LIN {X 0,Y 249.343,Z 705.614,A -85,B 0,C 180,E1 -25800.898,E2 -25800.898} C_VEL
LIN {X 0,Y 264.067,Z 715.978,A -85,B 0,C 180,E1 -25804.807,E2 -25804.807} C_VEL
LIN {X 0,Y 274.251,Z 722.94,A -85,B 0,C 180,E1 -25807.395,E2 -25807.395} C_VEL
LIN {X 0,Y 282.566,Z 728.902,A -85,B 0,C 180,E1 -25809.623,E2 -25809.623} C_VEL
LIN {X 0,Y 289.203,Z 733.495,A -85,B 0,C 180,E1 -25811.584,E2 -25811.584} C_VEL
LIN {X 0,Y 294.521,Z 737.29,A -85,B 0,C 180,E1 -25813.361,E2 -25813.361} C_VEL
LIN {X 0,Y 299.139,Z 740.278,A -85,B 0,C 180,E1 -25815.023,E2 -25815.023} C_VEL
LIN {X 0,Y 304.429,Z 743.64,A -85,B 0,C 180,E1 -25817.206,E2 -25817.206} C_VEL
LIN {X 0,Y 308.808,Z 746.666,A -85,B 0,C 180,E1 -25819.51,E2 -25819.51} C_VEL
LIN {X 0,Y 312.468,Z 748.873,A -85,B 0,C 180,E1 -25821.741,E2 -25821.741} C_VEL
LIN {X 0,Y 315.031,Z 750.212,A -85,B 0,C 180,E1 -25823.596,E2 -25823.596} C_VEL
LIN {X 0,Y 317.169,Z 751.257,A -85,B 0,C 180,E1 -25825.649,E2 -25825.649} C_VEL
LIN {X 0,Y 318.513,Z 751.721,A -85,B 0,C 180,E1 -25827.471,E2 -25827.471} C_VEL
LIN {X 0,Y 319.007,Z 751.919,A -85,B 0,C 180,E1 -25828.738,E2 -25828.738} C_VEL
LIN {X 0,Y 319.27,Z 751.929,A -85,B 0,C 180,E1 -25830,E2 -25830} C_VEL
LIN {X 0,Y 319.005,Z 751.919,A -85,B 0,C 180,E1 -25831.262,E2 -25831.262} C_VEL
LIN {X 0,Y 318.514,Z 751.721,A -85,B 0,C 180,E1 -25832.529,E2 -25832.529} C_VEL
LIN {X 0,Y 317.183,Z 751.226,A -85,B 0,C 180,E1 -25834.384,E2 -25834.384} C_VEL
LIN {X 0,Y 315.022,Z 750.196,A -85,B 0,C 180,E1 -25836.404,E2 -25836.404} C_VEL
LIN {X 0,Y 312.468,Z 748.905,A -85,B 0,C 180,E1 -25838.259,E2 -25838.259} C_VEL
LIN {X 0,Y 308.808,Z 746.698,A -85,B 0,C 180,E1 -25840.49,E2 -25840.49} C_VEL
LIN {X 0,Y 304.441,Z 743.645,A -85,B 0,C 180,E1 -25842.796,E2 -25842.796} C_VEL
LIN {X 0,Y 299.167,Z 740.269,A -85,B 0,C 180,E1 -25844.975,E2 -25844.975} C_VEL
LIN {X 0,Y 293.787,Z 736.797,A -85,B 0,C 180,E1 -25846.889,E2 -25846.889} C_VEL
LIN {X 0,Y 287.515,Z 732.243,A -85,B 0,C 180,E1 -25848.958,E2 -25848.958} C_VEL
LIN {X 0,Y 282.543,Z 728.898,A -85,B 0,C 180,E1 -25850.379,E2 -25850.379} C_VEL
LIN {X 0,Y 274.122,Z 722.857,A -85,B 0,C 180,E1 -25852.638,E2 -25852.638} C_VEL
LIN {X 0,Y 261.416,Z 714.087,A -85,B 0,C 180,E1 -25855.897,E2 -25855.897} C_VEL
LIN {X 0,Y 247.011,Z 703.927,A -85,B 0,C 180,E1 -25859.749,E2 -25859.749} C_VEL
LIN {X 0,Y 233.268,Z 692.779,A -85,B 0,C 180,E1 -25863.908,E2 -25863.908} C_VEL
LIN {X 0,Y 222.302,Z 681.729,A -85,B 0,C 180,E1 -25867.782,E2 -25867.782} C_VEL
LIN {X 0,Y 212.171,Z 669.521,A -85,B 0,C 180,E1 -25871.816,E2 -25871.816} C_VEL
LIN {X 0,Y 203.151,Z 656.416,A -85,B 0,C 180,E1 -25875.8,E2 -25875.8} C_VEL
LIN {X 0,Y 196.212,Z 644.549,A -85,B 0,C 180,E1 -25879.096,E2 -25879.096} C_VEL
LIN {X 0,Y 189.227,Z 630.541,A -85,B 0,C 180,E1 -25882.568,E2 -25882.568} C_VEL
LIN {X 0,Y 181.522,Z 611.257,A -85,B 0,C 180,E1 -25887.261,E2 -25887.261} C_VEL
LIN {X 0,Y 177.428,Z 602.179,A -85,B 0,C 180,E1 -25890.115,E2 -25890.115} C_VEL
LIN {X 0,Y 173.282,Z 594.104,A -85,B 0,C 180,E1 -25893.343,E2 -25893.343} C_VEL
LIN {X 0,Y 169.438,Z 587.347,A -85,B 0,C 180,E1 -25896.795,E2 -25896.795} C_VEL
LIN {X 0,Y 167.126,Z 583.517,A -85,B 0,C 180,E1 -25899.192,E2 -25899.192} C_VEL
LIN {X 0,Y 165.368,Z 580.676,A -85,B 0,C 180,E1 -25901.254,E2 -25901.254} C_VEL
LIN {X 0,Y 163.166,Z 577.17,A -85,B 0,C 180,E1 -25904.272,E2 -25904.272} C_VEL
LIN {X 0,Y 160.907,Z 573.312,A -85,B 0,C 180,E1 -25908.311,E2 -25908.311} C_VEL
LIN {X 0,Y 158.622,Z 569.898,A -85,B 0,C 180,E1 -25915.156,E2 -25915.156} C_VEL
LIN {X 0,Y 158.338,Z 568.536,A -85,B 0,C 180,E1 -25918.094,E2 -25918.094} C_VEL
LIN {X 0,Y 158.304,Z 568.373,A -85,B 0,C 180,E1 -25920.637,E2 -25920.637} C_VEL
LIN {X 0,Y 158.563,Z 569.545,A -85,B 0,C 180,E1 -25923.972,E2 -25923.972} C_VEL
LIN {X 0,Y 160.772,Z 573.178,A -85,B 0,C 180,E1 -25931.027,E2 -25931.027} C_VEL
LIN {X 0,Y 163.913,Z 578.324,A -85,B 0,C 180,E1 -25936.423,E2 -25936.423} C_VEL
LIN {X 0,Y 166.721,Z 582.763,A -85,B 0,C 180,E1 -25939.95,E2 -25939.95} C_VEL
LIN {X 0,Y 169.433,Z 587.305,A -85,B 0,C 180,E1 -25942.805,E2 -25942.805} C_VEL
LIN {X 0,Y 172.211,Z 592.35,A -85,B 0,C 180,E1 -25945.374,E2 -25945.374} C_VEL
LIN {X 0,Y 175.708,Z 601.255,A -85,B 0,C 180,E1 -25948.417,E2 -25948.417} C_VEL
LIN {X 0,Y 178.834,Z 610.413,A -85,B 0,C 180,E1 -25950.906,E2 -25950.906} C_VEL
LIN {X 0,Y 178.834,Z 612.491,A -85,B 0,C 180,E1 -25951.064,E2 -25951.064} C_VEL
LIN {X 0,Y 175.369,Z 650.601,A -85,B 0,C 180,E1 -25952.268,E2 -25952.268} C_VEL
LIN {X 0,Y 172.985,Z 664.836,A -85,B 0,C 180,E1 -25952.945,E2 -25952.945} C_VEL
LIN {X 0,Y 169.387,Z 678.905,A -85,B 0,C 180,E1 -25953.922,E2 -25953.922} C_VEL
LIN {X 0,Y 165.395,Z 691.016,A -85,B 0,C 180,E1 -25955.119,E2 -25955.119} C_VEL
LIN {X 0,Y 161.495,Z 700.931,A -85,B 0,C 180,E1 -25956.383,E2 -25956.383} C_VEL
LIN {X 0,Y 157.061,Z 710.649,A -85,B 0,C 180,E1 -25957.941,E2 -25957.941} C_VEL
LIN {X 0,Y 152.151,Z 720.062,A -85,B 0,C 180,E1 -25959.834,E2 -25959.834} C_VEL
LIN {X 0,Y 146.951,Z 729.125,A -85,B 0,C 180,E1 -25962.184,E2 -25962.184} C_VEL
LIN {X 0,Y 142.539,Z 736.054,A -85,B 0,C 180,E1 -25964.364,E2 -25964.364} C_VEL
LIN {X 0,Y 137.263,Z 743.572,A -85,B 0,C 180,E1 -25967.282,E2 -25967.282} C_VEL
LIN {X 0,Y 132.349,Z 750.042,A -85,B 0,C 180,E1 -25970.416,E2 -25970.416} C_VEL
LIN {X 0,Y 127.119,Z 756.583,A -85,B 0,C 180,E1 -25974.514,E2 -25974.514} C_VEL
LIN {X 0,Y 122.603,Z 762.018,A -85,B 0,C 180,E1 -25978.943,E2 -25978.943} C_VEL
LIN {X 0,Y 118.918,Z 766.47,A -85,B 0,C 180,E1 -25983.689,E2 -25983.689} C_VEL
LIN {X 0,Y 115.972,Z 770.022,A -85,B 0,C 180,E1 -25988.679,E2 -25988.679} C_VEL
LIN {X 0,Y 114.424,Z 771.967,A -85,B 0,C 180,E1 -25992.116,E2 -25992.116} C_VEL
LIN {X 0,Y 112.645,Z 774.671,A -85,B 0,C 180,E1 -25999.212,E2 -25999.212} C_VEL
LIN {X 0,Y 112.129,Z 775.98,A -85,B 0,C 180,E1 -26006.407,E2 -26006.407} C_VEL
LIN {X 0,Y 112.252,Z 776.239,A -85,B 0,C 180,E1 -26010,E2 -26010} C_VEL
LIN {X 0,Y 112.24,Z 775.497,A -85,B 0,C 180,E1 -26017.194,E2 -26017.194} C_VEL
LIN {X 0,Y 112.645,Z 774.671,A -85,B 0,C 180,E1 -26020.788,E2 -26020.788} C_VEL
LIN {X 0,Y 114.423,Z 771.967,A -85,B 0,C 180,E1 -26027.885,E2 -26027.885} C_VEL
LIN {X 0,Y 116.863,Z 769.003,A -85,B 0,C 180,E1 -26033.01,E2 -26033.01} C_VEL
LIN {X 0,Y 120.039,Z 765.169,A -85,B 0,C 180,E1 -26037.929,E2 -26037.929} C_VEL
LIN {X 0,Y 124.031,Z 760.401,A -85,B 0,C 180,E1 -26042.567,E2 -26042.567} C_VEL
LIN {X 0,Y 129.676,Z 753.456,A -85,B 0,C 180,E1 -26047.568,E2 -26047.568} C_VEL
LIN {X 0,Y 134.24,Z 747.582,A -85,B 0,C 180,E1 -26050.875,E2 -26050.875} C_VEL
LIN {X 0,Y 139.338,Z 740.737,A -85,B 0,C 180,E1 -26053.909,E2 -26053.909} C_VEL
LIN {X 0,Y 145.565,Z 731.458,A -85,B 0,C 180,E1 -26057.103,E2 -26057.103} C_VEL
LIN {X 0,Y 151.017,Z 722.182,A -85,B 0,C 180,E1 -26059.644,E2 -26059.644} C_VEL
LIN {X 0,Y 155.84,Z 713.129,A -85,B 0,C 180,E1 -26061.587,E2 -26061.587} C_VEL
LIN {X 0,Y 160.214,Z 703.858,A -85,B 0,C 180,E1 -26063.182,E2 -26063.182} C_VEL
LIN {X 0,Y 164.071,Z 694.521,A -85,B 0,C 180,E1 -26064.473,E2 -26064.473} C_VEL
LIN {X 0,Y 167.744,Z 684.271,A -85,B 0,C 180,E1 -26065.571,E2 -26065.571} C_VEL
LIN {X 0,Y 170.756,Z 673.982,A -85,B 0,C 180,E1 -26066.453,E2 -26066.453} C_VEL
LIN {X 0,Y 173.478,Z 662.099,A -85,B 0,C 180,E1 -26067.205,E2 -26067.205} C_VEL
LIN {X 0,Y 175.386,Z 650.33,A -85,B 0,C 180,E1 -26067.733,E2 -26067.733} C_VEL
LIN {X 0,Y 176.331,Z 641.978,A -85,B 0,C 180,E1 -26068.02,E2 -26068.02} C_VEL
LIN {X 0,Y 176.312,Z 638.104,A -85,B 0,C 180,E1 -26068.322,E2 -26068.322} C_VEL
LIN {X 0,Y 174.402,Z 626.17,A -85,B 0,C 180,E1 -26070.298,E2 -26070.298} C_VEL
LIN {X 0,Y 174.415,Z 622.295,A -85,B 0,C 180,E1 -26070.606,E2 -26070.606} C_VEL
LIN {X 0,Y 175.1,Z 613.268,A -85,B 0,C 180,E1 -26070.947,E2 -26070.947} C_VEL
LIN {X 0,Y 172.214,Z 604.583,A -85,B 0,C 180,E1 -26073.489,E2 -26073.489} C_VEL
LIN {X 0,Y 169.385,Z 597.046,A -85,B 0,C 180,E1 -26076.218,E2 -26076.218} C_VEL
LIN {X 0,Y 165.751,Z 590.516,A -85,B 0,C 180,E1 -26080.009,E2 -26080.009} C_VEL
LIN {X 0,Y 163.947,Z 587.5,A -85,B 0,C 180,E1 -26082.215,E2 -26082.215} C_VEL
LIN {X 0,Y 161.676,Z 583.716,A -85,B 0,C 180,E1 -26085.524,E2 -26085.524} C_VEL
LIN {X 0,Y 159.683,Z 580.121,A -85,B 0,C 180,E1 -26089.378,E2 -26089.378} C_VEL
LIN {X 0,Y 157.461,Z 575.531,A -85,B 0,C 180,E1 -26098.72,E2 -26098.72} C_VEL
LIN {X 0,Y 157.431,Z 575.384,A -85,B 0,C 180,E1 -26100.638,E2 -26100.638} C_VEL
LIN {X 0,Y 157.577,Z 576.308,A -85,B 0,C 180,E1 -26103.515,E2 -26103.515} C_VEL
LIN {X 0,Y 159.657,Z 580.101,A -85,B 0,C 180,E1 -26110.961,E2 -26110.961} C_VEL
LIN {X 0,Y 162.611,Z 585.221,A -85,B 0,C 180,E1 -26116.314,E2 -26116.314} C_VEL
LIN {X 0,Y 164.955,Z 589.145,A -85,B 0,C 180,E1 -26119.441,E2 -26119.441} C_VEL
LIN {X 0,Y 168.312,Z 595.05,A -85,B 0,C 180,E1 -26123.127,E2 -26123.127} C_VEL
LIN {X 0,Y 172.251,Z 602.608,A -85,B 0,C 180,E1 -26126.748,E2 -26126.748} C_VEL
LIN {X 0,Y 176.372,Z 611.496,A -85,B 0,C 180,E1 -26130.034,E2 -26130.034} C_VEL
LIN {X 0,Y 180.211,Z 621.162,A -85,B 0,C 180,E1 -26132.804,E2 -26132.804} C_VEL
LIN {X 0,Y 186.639,Z 637.619,A -85,B 0,C 180,E1 -26136.823,E2 -26136.823} C_VEL
LIN {X 0,Y 193.199,Z 651.318,A -85,B 0,C 180,E1 -26140.47,E2 -26140.47} C_VEL
LIN {X 0,Y 199.834,Z 663.107,A -85,B 0,C 180,E1 -26143.993,E2 -26143.993} C_VEL
LIN {X 0,Y 206.871,Z 673.757,A -85,B 0,C 180,E1 -26147.454,E2 -26147.454} C_VEL
LIN {X 0,Y 215.839,Z 684.961,A -85,B 0,C 180,E1 -26151.394,E2 -26151.394} C_VEL
LIN {X 0,Y 224.654,Z 694.377,A -85,B 0,C 180,E1 -26154.852,E2 -26154.852} C_VEL
LIN {X 0,Y 234.457,Z 702.998,A -85,B 0,C 180,E1 -26158.209,E2 -26158.209} C_VEL
LIN {X 0,Y 248.506,Z 713.424,A -85,B 0,C 180,E1 -26162.414,E2 -26162.414} C_VEL
LIN {X 0,Y 259.962,Z 721.098,A -85,B 0,C 180,E1 -26165.528,E2 -26165.528} C_VEL
LIN {X 0,Y 270.032,Z 727.797,A -85,B 0,C 180,E1 -26168.198,E2 -26168.198} C_VEL
LIN {X 0,Y 280.047,Z 734.699,A -85,B 0,C 180,E1 -26170.959,E2 -26170.959} C_VEL
LIN {X 0,Y 286.565,Z 739.311,A -85,B 0,C 180,E1 -26173.03,E2 -26173.03} C_VEL
LIN {X 0,Y 292.618,Z 743.324,A -85,B 0,C 180,E1 -26175.152,E2 -26175.152} C_VEL
LIN {X 0,Y 296.251,Z 745.63,A -85,B 0,C 180,E1 -26176.565,E2 -26176.565} C_VEL
LIN {X 0,Y 298.933,Z 747.459,A -85,B 0,C 180,E1 -26177.785,E2 -26177.785} C_VEL
LIN {X 0,Y 301.745,Z 749.392,A -85,B 0,C 180,E1 -26179.262,E2 -26179.262} C_VEL
LIN {X 0,Y 305.564,Z 751.769,A -85,B 0,C 180,E1 -26181.49,E2 -26181.49} C_VEL
LIN {X 0,Y 308.374,Z 753.28,A -85,B 0,C 180,E1 -26183.457,E2 -26183.457} C_VEL
LIN {X 0,Y 310.322,Z 754.209,A -85,B 0,C 180,E1 -26185.187,E2 -26185.187} C_VEL
LIN {X 0,Y 311.213,Z 754.584,A -85,B 0,C 180,E1 -26186.115,E2 -26186.115} C_VEL
LIN {X 0,Y 312.139,Z 754.94,A -85,B 0,C 180,E1 -26187.419,E2 -26187.419} C_VEL
LIN {X 0,Y 312.683,Z 755.143,A -85,B 0,C 180,E1 -26188.712,E2 -26188.712} C_VEL
LIN {X 0,Y 312.947,Z 755.169,A -85,B 0,C 180,E1 -26190,E2 -26190} C_VEL
LIN {X 0,Y 312.681,Z 755.141,A -85,B 0,C 180,E1 -26191.288,E2 -26191.288} C_VEL
LIN {X 0,Y 312.138,Z 754.937,A -85,B 0,C 180,E1 -26192.581,E2 -26192.581} C_VEL
LIN {X 0,Y 310.329,Z 754.212,A -85,B 0,C 180,E1 -26194.83,E2 -26194.83} C_VEL
LIN {X 0,Y 308.364,Z 753.256,A -85,B 0,C 180,E1 -26196.543,E2 -26196.543} C_VEL
LIN {X 0,Y 305.57,Z 751.76,A -85,B 0,C 180,E1 -26198.519,E2 -26198.519} C_VEL
LIN {X 0,Y 300.901,Z 748.83,A -85,B 0,C 180,E1 -26201.199,E2 -26201.199} C_VEL
LIN {X 0,Y 298.945,Z 747.432,A -85,B 0,C 180,E1 -26202.215,E2 -26202.215} C_VEL
LIN {X 0,Y 295.517,Z 745.126,A -85,B 0,C 180,E1 -26203.758,E2 -26203.758} C_VEL
LIN {X 0,Y 289.867,Z 741.603,A -85,B 0,C 180,E1 -26205.837,E2 -26205.837} C_VEL
LIN {X 0,Y 283.245,Z 736.916,A -85,B 0,C 180,E1 -26208.091,E2 -26208.091} C_VEL
LIN {X 0,Y 276.681,Z 732.425,A -85,B 0,C 180,E1 -26209.978,E2 -26209.978} C_VEL
LIN {X 0,Y 268.367,Z 726.639,A -85,B 0,C 180,E1 -26212.263,E2 -26212.263} C_VEL
LIN {X 0,Y 256.678,Z 718.841,A -85,B 0,C 180,E1 -26215.372,E2 -26215.372} C_VEL
LIN {X 0,Y 241.269,Z 708.265,A -85,B 0,C 180,E1 -26219.682,E2 -26219.682} C_VEL
LIN {X 0,Y 227.281,Z 696.899,A -85,B 0,C 180,E1 -26224.193,E2 -26224.193} C_VEL
LIN {X 0,Y 217.681,Z 687.148,A -85,B 0,C 180,E1 -26227.837,E2 -26227.837} C_VEL
LIN {X 0,Y 209.331,Z 676.985,A -85,B 0,C 180,E1 -26231.427,E2 -26231.427} C_VEL
LIN {X 0,Y 202.538,Z 667.322,A -85,B 0,C 180,E1 -26234.657,E2 -26234.657} C_VEL
LIN {X 0,Y 195.897,Z 656.31,A -85,B 0,C 180,E1 -26238.069,E2 -26238.069} C_VEL
LIN {X 0,Y 190.345,Z 645.491,A -85,B 0,C 180,E1 -26241.122,E2 -26241.122} C_VEL
LIN {X 0,Y 184.465,Z 632.548,A -85,B 0,C 180,E1 -26244.428,E2 -26244.428} C_VEL
LIN {X 0,Y 178.246,Z 615.988,A -85,B 0,C 180,E1 -26248.589,E2 -26248.589} C_VEL
LIN {X 0,Y 174.561,Z 607.48,A -85,B 0,C 180,E1 -26251.358,E2 -26251.358} C_VEL
LIN {X 0,Y 170.911,Z 599.958,A -85,B 0,C 180,E1 -26254.419,E2 -26254.419} C_VEL
LIN {X 0,Y 167.054,Z 592.841,A -85,B 0,C 180,E1 -26258.167,E2 -26258.167} C_VEL
LIN {X 0,Y 164.13,Z 587.743,A -85,B 0,C 180,E1 -26261.593,E2 -26261.593} C_VEL
LIN {X 0,Y 161.728,Z 583.787,A -85,B 0,C 180,E1 -26265.049,E2 -26265.049} C_VEL
LIN {X 0,Y 159.558,Z 580.057,A -85,B 0,C 180,E1 -26269.239,E2 -26269.239} C_VEL
LIN {X 0,Y 157.469,Z 575.62,A -85,B 0,C 180,E1 -26278.083,E2 -26278.083} C_VEL
LIN {X 0,Y 157.438,Z 575.431,A -85,B 0,C 180,E1 -26280.641,E2 -26280.641} C_VEL
LIN {X 0,Y 157.623,Z 576.478,A -85,B 0,C 180,E1 -26283.516,E2 -26283.516} C_VEL
LIN {X 0,Y 159.886,Z 580.526,A -85,B 0,C 180,E1 -26291.089,E2 -26291.089} C_VEL
LIN {X 0,Y 162.452,Z 584.977,A -85,B 0,C 180,E1 -26295.688,E2 -26295.688} C_VEL
LIN {X 0,Y 165.069,Z 589.338,A -85,B 0,C 180,E1 -26299.187,E2 -26299.187} C_VEL
LIN {X 0,Y 168.093,Z 594.615,A -85,B 0,C 180,E1 -26302.51,E2 -26302.51} C_VEL
LIN {X 0,Y 169.951,Z 598.44,A -85,B 0,C 180,E1 -26304.347,E2 -26304.347} C_VEL
LIN {X 0,Y 173.054,Z 607.008,A -85,B 0,C 180,E1 -26307.273,E2 -26307.273} C_VEL
LIN {X 0,Y 175.104,Z 613.293,A -85,B 0,C 180,E1 -26309.058,E2 -26309.058} C_VEL
LIN {X 0,Y 172.897,Z 639.291,A -85,B 0,C 180,E1 -26309.905,E2 -26309.905} C_VEL
LIN {X 0,Y 170.844,Z 656.23,A -85,B 0,C 180,E1 -26310.507,E2 -26310.507} C_VEL
LIN {X 0,Y 168.29,Z 668.57,A -85,B 0,C 180,E1 -26311.168,E2 -26311.168} C_VEL
LIN {X 0,Y 165.182,Z 679.779,A -85,B 0,C 180,E1 -26311.977,E2 -26311.977} C_VEL
LIN {X 0,Y 161.404,Z 690.818,A -85,B 0,C 180,E1 -26313.052,E2 -26313.052} C_VEL
LIN {X 0,Y 157.387,Z 700.733,A -85,B 0,C 180,E1 -26314.302,E2 -26314.302} C_VEL
LIN {X 0,Y 152.795,Z 710.451,A -85,B 0,C 180,E1 -26315.839,E2 -26315.839} C_VEL
LIN {X 0,Y 147.696,Z 719.863,A -85,B 0,C 180,E1 -26317.714,E2 -26317.714} C_VEL
LIN {X 0,Y 142.813,Z 728.023,A -85,B 0,C 180,E1 -26319.775,E2 -26319.775} C_VEL
LIN {X 0,Y 137.633,Z 735.854,A -85,B 0,C 180,E1 -26322.234,E2 -26322.234} C_VEL
LIN {X 0,Y 132.114,Z 743.374,A -85,B 0,C 180,E1 -26325.183,E2 -26325.183} C_VEL
LIN {X 0,Y 126.909,Z 749.843,A -85,B 0,C 180,E1 -26328.354,E2 -26328.354} C_VEL
LIN {X 0,Y 121.375,Z 756.383,A -85,B 0,C 180,E1 -26332.557,E2 -26332.557} C_VEL
LIN {X 0,Y 116.524,Z 761.818,A -85,B 0,C 180,E1 -26337.125,E2 -26337.125} C_VEL
LIN {X 0,Y 112.55,Z 766.27,A -85,B 0,C 180,E1 -26342.075,E2 -26342.075} C_VEL
LIN {X 0,Y 109.341,Z 769.822,A -85,B 0,C 180,E1 -26347.316,E2 -26347.316} C_VEL
LIN {X 0,Y 107.64,Z 771.767,A -85,B 0,C 180,E1 -26350.946,E2 -26350.946} C_VEL
LIN {X 0,Y 105.636,Z 774.471,A -85,B 0,C 180,E1 -26358.487,E2 -26358.487} C_VEL
LIN {X 0,Y 105.036,Z 775.781,A -85,B 0,C 180,E1 -26366.164,E2 -26366.164} C_VEL
LIN {X 0,Y 105.17,Z 776.042,A -85,B 0,C 180,E1 -26370,E2 -26370} C_VEL
LIN {X 0,Y 105.175,Z 775.299,A -85,B 0,C 180,E1 -26377.68,E2 -26377.68} C_VEL
LIN {X 0,Y 105.636,Z 774.471,A -85,B 0,C 180,E1 -26381.513,E2 -26381.513} C_VEL
LIN {X 0,Y 107.639,Z 771.767,A -85,B 0,C 180,E1 -26389.054,E2 -26389.054} C_VEL
LIN {X 0,Y 110.319,Z 768.804,A -85,B 0,C 180,E1 -26394.461,E2 -26394.461} C_VEL
LIN {X 0,Y 114.989,Z 763.502,A -85,B 0,C 180,E1 -26401.164,E2 -26401.164} C_VEL
LIN {X 0,Y 119.675,Z 758.297,A -85,B 0,C 180,E1 -26405.962,E2 -26405.962} C_VEL
LIN {X 0,Y 125.011,Z 752.119,A -85,B 0,C 180,E1 -26410.279,E2 -26410.279} C_VEL
LIN {X 0,Y 129.955,Z 746.046,A -85,B 0,C 180,E1 -26413.591,E2 -26413.591} C_VEL
LIN {X 0,Y 135.408,Z 738.978,A -85,B 0,C 180,E1 -26416.604,E2 -26416.604} C_VEL
LIN {X 0,Y 139.995,Z 732.521,A -85,B 0,C 180,E1 -26418.852,E2 -26418.852} C_VEL
LIN {X 0,Y 145.902,Z 723.043,A -85,B 0,C 180,E1 -26421.512,E2 -26421.512} C_VEL
LIN {X 0,Y 150.886,Z 714.17,A -85,B 0,C 180,E1 -26423.461,E2 -26423.461} C_VEL
LIN {X 0,Y 155.409,Z 705.124,A -85,B 0,C 180,E1 -26425.049,E2 -26425.049} C_VEL
LIN {X 0,Y 160.05,Z 694.323,A -85,B 0,C 180,E1 -26426.543,E2 -26426.543} C_VEL
LIN {X 0,Y 163.841,Z 684.073,A -85,B 0,C 180,E1 -26427.616,E2 -26427.616} C_VEL
LIN {X 0,Y 167.251,Z 672.563,A -85,B 0,C 180,E1 -26428.568,E2 -26428.568} C_VEL
LIN {X 0,Y 169.814,Z 661.454,A -85,B 0,C 180,E1 -26429.247,E2 -26429.247} C_VEL
LIN {X 0,Y 171.692,Z 650.197,A -85,B 0,C 180,E1 -26429.735,E2 -26429.735} C_VEL
LIN {X 0,Y 174.415,Z 622.295,A -85,B 0,C 180,E1 -26430.606,E2 -26430.606} C_VEL
LIN {X 0,Y 174.31,Z 619.282,A -85,B 0,C 180,E1 -26430.914,E2 -26430.914} C_VEL
LIN {X 0,Y 173.654,Z 616.695,A -85,B 0,C 180,E1 -26431.52,E2 -26431.52} C_VEL
LIN {X 0,Y 172.484,Z 614.168,A -85,B 0,C 180,E1 -26432.459,E2 -26432.459} C_VEL
LIN {X 0,Y 169.273,Z 608.739,A -85,B 0,C 180,E1 -26435.131,E2 -26435.131} C_VEL
LIN {X 0,Y 168.904,Z 607.826,A -85,B 0,C 180,E1 -26435.49,E2 -26435.49} C_VEL
LIN {X 0,Y 166.942,Z 602.523,A -85,B 0,C 180,E1 -26437.571,E2 -26437.571} C_VEL
LIN {X 0,Y 163.858,Z 596.656,A -85,B 0,C 180,E1 -26441.072,E2 -26441.072} C_VEL
LIN {X 0,Y 162.062,Z 593.514,A -85,B 0,C 180,E1 -26443.464,E2 -26443.464} C_VEL
LIN {X 0,Y 160.334,Z 590.422,A -85,B 0,C 180,E1 -26446.21,E2 -26446.21} C_VEL
LIN {X 0,Y 158.463,Z 586.917,A -85,B 0,C 180,E1 -26450.103,E2 -26450.103} C_VEL
LIN {X 0,Y 156.591,Z 582.617,A -85,B 0,C 180,E1 -26458.713,E2 -26458.713} C_VEL
LIN {X 0,Y 156.566,Z 582.432,A -85,B 0,C 180,E1 -26460.642,E2 -26460.642} C_VEL
LIN {X 0,Y 156.67,Z 583.317,A -85,B 0,C 180,E1 -26463.213,E2 -26463.213} C_VEL
LIN {X 0,Y 158.726,Z 587.386,A -85,B 0,C 180,E1 -26470.923,E2 -26470.923} C_VEL
LIN {X 0,Y 161.217,Z 591.969,A -85,B 0,C 180,E1 -26475.647,E2 -26475.647} C_VEL
LIN {X 0,Y 163.355,Z 595.768,A -85,B 0,C 180,E1 -26478.685,E2 -26478.685} C_VEL
LIN {X 0,Y 166.273,Z 601.159,A -85,B 0,C 180,E1 -26482.107,E2 -26482.107} C_VEL
LIN {X 0,Y 170.28,Z 609.336,A -85,B 0,C 180,E1 -26486.033,E2 -26486.033} C_VEL
LIN {X 0,Y 173.891,Z 617.792,A -85,B 0,C 180,E1 -26489.107,E2 -26489.107} C_VEL
LIN {X 0,Y 177.053,Z 626.293,A -85,B 0,C 180,E1 -26491.564,E2 -26491.564} C_VEL
LIN {X 0,Y 182.955,Z 642.316,A -85,B 0,C 180,E1 -26495.636,E2 -26495.636} C_VEL
LIN {X 0,Y 187.829,Z 653.466,A -85,B 0,C 180,E1 -26498.739,E2 -26498.739} C_VEL
LIN {X 0,Y 192.706,Z 663.195,A -85,B 0,C 180,E1 -26501.725,E2 -26501.725} C_VEL
LIN {X 0,Y 198.541,Z 673.231,A -85,B 0,C 180,E1 -26505.068,E2 -26505.068} C_VEL
LIN {X 0,Y 205.646,Z 683.514,A -85,B 0,C 180,E1 -26508.75,E2 -26508.75} C_VEL
LIN {X 0,Y 215.102,Z 694.784,A -85,B 0,C 180,E1 -26513.058,E2 -26513.058} C_VEL
LIN {X 0,Y 225.755,Z 704.956,A -85,B 0,C 180,E1 -26517.195,E2 -26517.195} C_VEL
LIN {X 0,Y 239.524,Z 715.344,A -85,B 0,C 180,E1 -26521.67,E2 -26521.67} C_VEL
LIN {X 0,Y 252.118,Z 723.619,A -85,B 0,C 180,E1 -26525.284,E2 -26525.284} C_VEL
LIN {X 0,Y 264.183,Z 731.336,A -85,B 0,C 180,E1 -26528.604,E2 -26528.604} C_VEL
LIN {X 0,Y 274.26,Z 738.006,A -85,B 0,C 180,E1 -26531.463,E2 -26531.463} C_VEL
LIN {X 0,Y 281.399,Z 743.034,A -85,B 0,C 180,E1 -26533.734,E2 -26533.734} C_VEL
LIN {X 0,Y 287.297,Z 746.886,A -85,B 0,C 180,E1 -26535.841,E2 -26535.841} C_VEL
LIN {X 0,Y 291.26,Z 749.46,A -85,B 0,C 180,E1 -26537.458,E2 -26537.458} C_VEL
LIN {X 0,Y 294.436,Z 751.63,A -85,B 0,C 180,E1 -26538.992,E2 -26538.992} C_VEL
LIN {X 0,Y 298.569,Z 754.255,A -85,B 0,C 180,E1 -26541.348,E2 -26541.348} C_VEL
LIN {X 0,Y 301.468,Z 755.905,A -85,B 0,C 180,E1 -26543.306,E2 -26543.306} C_VEL
LIN {X 0,Y 303.4,Z 756.816,A -85,B 0,C 180,E1 -26544.9,E2 -26544.9} C_VEL
LIN {X 0,Y 304.532,Z 757.314,A -85,B 0,C 180,E1 -26546.03,E2 -26546.03} C_VEL
LIN {X 0,Y 305.54,Z 757.724,A -85,B 0,C 180,E1 -26547.363,E2 -26547.363} C_VEL
LIN {X 0,Y 306.138,Z 757.962,A -85,B 0,C 180,E1 -26548.685,E2 -26548.685} C_VEL
LIN {X 0,Y 306.436,Z 757.996,A -85,B 0,C 180,E1 -26550,E2 -26550} C_VEL
LIN {X 0,Y 306.136,Z 757.958,A -85,B 0,C 180,E1 -26551.315,E2 -26551.315} C_VEL
LIN {X 0,Y 305.54,Z 757.717,A -85,B 0,C 180,E1 -26552.637,E2 -26552.637} C_VEL
LIN {X 0,Y 304.539,Z 757.299,A -85,B 0,C 180,E1 -26553.97,E2 -26553.97} C_VEL
LIN {X 0,Y 303.157,Z 756.7,A -85,B 0,C 180,E1 -26555.321,E2 -26555.321} C_VEL
LIN {X 0,Y 301.457,Z 755.888,A -85,B 0,C 180,E1 -26556.694,E2 -26556.694} C_VEL
LIN {X 0,Y 298.573,Z 754.251,A -85,B 0,C 180,E1 -26558.657,E2 -26558.657} C_VEL
LIN {X 0,Y 293.848,Z 751.22,A -85,B 0,C 180,E1 -26561.309,E2 -26561.309} C_VEL
LIN {X 0,Y 289.102,Z 747.988,A -85,B 0,C 180,E1 -26563.499,E2 -26563.499} C_VEL
LIN {X 0,Y 282.522,Z 743.805,A -85,B 0,C 180,E1 -26565.88,E2 -26565.88} C_VEL
LIN {X 0,Y 277.007,Z 739.833,A -85,B 0,C 180,E1 -26567.725,E2 -26567.725} C_VEL
LIN {X 0,Y 269.191,Z 734.697,A -85,B 0,C 180,E1 -26569.971,E2 -26569.971} C_VEL
LIN {X 0,Y 261.624,Z 729.69,A -85,B 0,C 180,E1 -26572.091,E2 -26572.091} C_VEL
LIN {X 0,Y 249.205,Z 721.757,A -85,B 0,C 180,E1 -26575.52,E2 -26575.52} C_VEL
LIN {X 0,Y 234.812,Z 712.009,A -85,B 0,C 180,E1 -26579.777,E2 -26579.777} C_VEL
LIN {X 0,Y 223.585,Z 703.071,A -85,B 0,C 180,E1 -26583.596,E2 -26583.596} C_VEL
LIN {X 0,Y 212.297,Z 691.665,A -85,B 0,C 180,E1 -26588.167,E2 -26588.167} C_VEL
LIN {X 0,Y 202.026,Z 678.57,A -85,B 0,C 180,E1 -26593.07,E2 -26593.07} C_VEL
LIN {X 0,Y 195.156,Z 667.699,A -85,B 0,C 180,E1 -26596.826,E2 -26596.826} C_VEL
LIN {X 0,Y 188.992,Z 655.999,A -85,B 0,C 180,E1 -26600.524,E2 -26600.524} C_VEL
LIN {X 0,Y 183.42,Z 643.374,A -85,B 0,C 180,E1 -26604.103,E2 -26604.103} C_VEL
LIN {X 0,Y 175.122,Z 620.901,A -85,B 0,C 180,E1 -26609.92,E2 -26609.92} C_VEL
LIN {X 0,Y 171.908,Z 613.017,A -85,B 0,C 180,E1 -26612.537,E2 -26612.537} C_VEL
LIN {X 0,Y 168.575,Z 605.761,A -85,B 0,C 180,E1 -26615.551,E2 -26615.551} C_VEL
LIN {X 0,Y 164.934,Z 598.64,A -85,B 0,C 180,E1 -26619.385,E2 -26619.385} C_VEL
LIN {X 0,Y 162.232,Z 593.761,A -85,B 0,C 180,E1 -26622.836,E2 -26622.836} C_VEL
LIN {X 0,Y 160.43,Z 590.565,A -85,B 0,C 180,E1 -26625.655,E2 -26625.655} C_VEL
LIN {X 0,Y 158.427,Z 586.931,A -85,B 0,C 180,E1 -26629.78,E2 -26629.78} C_VEL
LIN {X 0,Y 156.599,Z 582.705,A -85,B 0,C 180,E1 -26638.072,E2 -26638.072} C_VEL
LIN {X 0,Y 156.571,Z 582.488,A -85,B 0,C 180,E1 -26640.644,E2 -26640.644} C_VEL
LIN {X 0,Y 156.738,Z 583.696,A -85,B 0,C 180,E1 -26643.536,E2 -26643.536} C_VEL
LIN {X 0,Y 158.726,Z 587.364,A -85,B 0,C 180,E1 -26650.525,E2 -26650.525} C_VEL
LIN {X 0,Y 161.064,Z 591.729,A -85,B 0,C 180,E1 -26655.017,E2 -26655.017} C_VEL
LIN {X 0,Y 163.36,Z 595.761,A -85,B 0,C 180,E1 -26658.297,E2 -26658.297} C_VEL
LIN {X 0,Y 166.071,Z 600.746,A -85,B 0,C 180,E1 -26661.493,E2 -26661.493} C_VEL
LIN {X 0,Y 167.75,Z 604.501,A -85,B 0,C 180,E1 -26663.291,E2 -26663.291} C_VEL
LIN {X 0,Y 170.89,Z 613.943,A -85,B 0,C 180,E1 -26666.486,E2 -26666.486} C_VEL
LIN {X 0,Y 171.548,Z 616.124,A -85,B 0,C 180,E1 -26667.115,E2 -26667.115} C_VEL
LIN {X 0,Y 168.204,Z 650.359,A -85,B 0,C 180,E1 -26668.183,E2 -26668.183} C_VEL
LIN {X 0,Y 165.58,Z 665.008,A -85,B 0,C 180,E1 -26668.849,E2 -26668.849} C_VEL
LIN {X 0,Y 161.54,Z 679.582,A -85,B 0,C 180,E1 -26669.844,E2 -26669.844} C_VEL
LIN {X 0,Y 157.648,Z 690.62,A -85,B 0,C 180,E1 -26670.89,E2 -26670.89} C_VEL
LIN {X 0,Y 153.499,Z 700.535,A -85,B 0,C 180,E1 -26672.112,E2 -26672.112} C_VEL
LIN {X 0,Y 148.739,Z 710.252,A -85,B 0,C 180,E1 -26673.615,E2 -26673.615} C_VEL
LIN {X 0,Y 143.44,Z 719.664,A -85,B 0,C 180,E1 -26675.458,E2 -26675.458} C_VEL
LIN {X 0,Y 137.88,Z 728.532,A -85,B 0,C 180,E1 -26677.711,E2 -26677.711} C_VEL
LIN {X 0,Y 132.941,Z 735.655,A -85,B 0,C 180,E1 -26679.956,E2 -26679.956} C_VEL
LIN {X 0,Y 127.137,Z 743.174,A -85,B 0,C 180,E1 -26682.91,E2 -26682.91} C_VEL
LIN {X 0,Y 121.657,Z 749.643,A -85,B 0,C 180,E1 -26686.115,E2 -26686.115} C_VEL
LIN {X 0,Y 115.781,Z 756.184,A -85,B 0,C 180,E1 -26690.406,E2 -26690.406} C_VEL
LIN {X 0,Y 110.59,Z 761.619,A -85,B 0,C 180,E1 -26695.114,E2 -26695.114} C_VEL
LIN {X 0,Y 106.285,Z 766.071,A -85,B 0,C 180,E1 -26700.27,E2 -26700.27} C_VEL
LIN {X 0,Y 102.786,Z 769.623,A -85,B 0,C 180,E1 -26705.78,E2 -26705.78} C_VEL
LIN {X 0,Y 100.907,Z 771.568,A -85,B 0,C 180,E1 -26709.621,E2 -26709.621} C_VEL
LIN {X 0,Y 98.659,Z 774.273,A -85,B 0,C 180,E1 -26717.661,E2 -26717.661} C_VEL
LIN {X 0,Y 97.939,Z 775.583,A -85,B 0,C 180,E1 -26725.885,E2 -26725.885} C_VEL
LIN {X 0,Y 98.076,Z 775.844,A -85,B 0,C 180,E1 -26730,E2 -26730} C_VEL
LIN {X 0,Y 98.113,Z 775.1,A -85,B 0,C 180,E1 -26738.237,E2 -26738.237} C_VEL
LIN {X 0,Y 98.659,Z 774.273,A -85,B 0,C 180,E1 -26742.339,E2 -26742.339} C_VEL
LIN {X 0,Y 100.905,Z 771.568,A -85,B 0,C 180,E1 -26750.38,E2 -26750.38} C_VEL
LIN {X 0,Y 103.842,Z 768.604,A -85,B 0,C 180,E1 -26756.098,E2 -26756.098} C_VEL
LIN {X 0,Y 108.508,Z 763.74,A -85,B 0,C 180,E1 -26762.645,E2 -26762.645} C_VEL
LIN {X 0,Y 113.956,Z 758.097,A -85,B 0,C 180,E1 -26768.077,E2 -26768.077} C_VEL
LIN {X 0,Y 119.655,Z 751.92,A -85,B 0,C 180,E1 -26772.489,E2 -26772.489} C_VEL
LIN {X 0,Y 124.891,Z 745.847,A -85,B 0,C 180,E1 -26775.846,E2 -26775.846} C_VEL
LIN {X 0,Y 130.61,Z 738.779,A -85,B 0,C 180,E1 -26778.878,E2 -26778.878} C_VEL
LIN {X 0,Y 136.399,Z 730.885,A -85,B 0,C 180,E1 -26781.541,E2 -26781.541} C_VEL
LIN {X 0,Y 142.19,Z 721.784,A -85,B 0,C 180,E1 -26784.032,E2 -26784.032} C_VEL
LIN {X 0,Y 147.418,Z 712.732,A -85,B 0,C 180,E1 -26785.926,E2 -26785.926} C_VEL
LIN {X 0,Y 152.11,Z 703.461,A -85,B 0,C 180,E1 -26787.478,E2 -26787.478} C_VEL
LIN {X 0,Y 156.244,Z 694.125,A -85,B 0,C 180,E1 -26788.717,E2 -26788.717} C_VEL
LIN {X 0,Y 160.143,Z 683.875,A -85,B 0,C 180,E1 -26789.767,E2 -26789.767} C_VEL
LIN {X 0,Y 163.568,Z 672.726,A -85,B 0,C 180,E1 -26790.663,E2 -26790.663} C_VEL
LIN {X 0,Y 166.227,Z 661.622,A -85,B 0,C 180,E1 -26791.33,E2 -26791.33} C_VEL
LIN {X 0,Y 168.23,Z 650.049,A -85,B 0,C 180,E1 -26791.815,E2 -26791.815} C_VEL
LIN {X 0,Y 171.543,Z 616.171,A -85,B 0,C 180,E1 -26792.884,E2 -26792.884} C_VEL
LIN {X 0,Y 168.904,Z 607.826,A -85,B 0,C 180,E1 -26795.49,E2 -26795.49} C_VEL
LIN {X 0,Y 167.839,Z 605.596,A -85,B 0,C 180,E1 -26796.525,E2 -26796.525} C_VEL
LIN {X 0,Y 165.977,Z 603.346,A -85,B 0,C 180,E1 -26798.291,E2 -26798.291} C_VEL
LIN {X 0,Y 162.796,Z 601.308,A -85,B 0,C 180,E1 -26801.542,E2 -26801.542} C_VEL
LIN {X 0,Y 160.137,Z 599.18,A -85,B 0,C 180,E1 -26804.955,E2 -26804.955} C_VEL
LIN {X 0,Y 159.723,Z 598.508,A -85,B 0,C 180,E1 -26805.628,E2 -26805.628} C_VEL
LIN {X 0,Y 158.523,Z 596.35,A -85,B 0,C 180,E1 -26807.842,E2 -26807.842} C_VEL
LIN {X 0,Y 157.335,Z 593.765,A -85,B 0,C 180,E1 -26810.68,E2 -26810.68} C_VEL
LIN {X 0,Y 155.707,Z 589.528,A -85,B 0,C 180,E1 -26819.352,E2 -26819.352} C_VEL
LIN {X 0,Y 155.717,Z 589.698,A -85,B 0,C 180,E1 -26821.615,E2 -26821.615} C_VEL
LIN {X 0,Y 157.588,Z 594.287,A -85,B 0,C 180,E1 -26830.379,E2 -26830.379} C_VEL
LIN {X 0,Y 159.717,Z 598.395,A -85,B 0,C 180,E1 -26834.736,E2 -26834.736} C_VEL
LIN {X 0,Y 161.861,Z 602.537,A -85,B 0,C 180,E1 -26838.02,E2 -26838.02} C_VEL
LIN {X 0,Y 164.608,Z 608.014,A -85,B 0,C 180,E1 -26841.442,E2 -26841.442} C_VEL
LIN {X 0,Y 167.774,Z 614.812,A -85,B 0,C 180,E1 -26844.764,E2 -26844.764} C_VEL
LIN {X 0,Y 171.007,Z 622.869,A -85,B 0,C 180,E1 -26847.761,E2 -26847.761} C_VEL
LIN {X 0,Y 173.831,Z 630.857,A -85,B 0,C 180,E1 -26850.148,E2 -26850.148} C_VEL
LIN {X 0,Y 178.567,Z 644.992,A -85,B 0,C 180,E1 -26853.854,E2 -26853.854} C_VEL
LIN {X 0,Y 182.278,Z 654.564,A -85,B 0,C 180,E1 -26856.62,E2 -26856.62} C_VEL
LIN {X 0,Y 185.925,Z 663.197,A -85,B 0,C 180,E1 -26859.282,E2 -26859.282} C_VEL
LIN {X 0,Y 191.704,Z 674.574,A -85,B 0,C 180,E1 -26863.186,E2 -26863.186} C_VEL
LIN {X 0,Y 197.684,Z 684.259,A -85,B 0,C 180,E1 -26866.785,E2 -26866.785} C_VEL
LIN {X 0,Y 204.913,Z 693.824,A -85,B 0,C 180,E1 -26870.596,E2 -26870.596} C_VEL
LIN {X 0,Y 213.49,Z 703.305,A -85,B 0,C 180,E1 -26874.562,E2 -26874.562} C_VEL
LIN {X 0,Y 223.025,Z 711.686,A -85,B 0,C 180,E1 -26878.3,E2 -26878.3} C_VEL
LIN {X 0,Y 236.874,Z 721.516,A -85,B 0,C 180,E1 -26882.883,E2 -26882.883} C_VEL
LIN {X 0,Y 247.884,Z 728.415,A -85,B 0,C 180,E1 -26886.121,E2 -26886.121} C_VEL
LIN {X 0,Y 259.347,Z 735.421,A -85,B 0,C 180,E1 -26889.373,E2 -26889.373} C_VEL
LIN {X 0,Y 269.288,Z 741.658,A -85,B 0,C 180,E1 -26892.282,E2 -26892.282} C_VEL
LIN {X 0,Y 274.563,Z 745.246,A -85,B 0,C 180,E1 -26893.973,E2 -26893.973} C_VEL
LIN {X 0,Y 281.827,Z 750.023,A -85,B 0,C 180,E1 -26896.542,E2 -26896.542} C_VEL
LIN {X 0,Y 286.722,Z 753.247,A -85,B 0,C 180,E1 -26898.692,E2 -26898.692} C_VEL
LIN {X 0,Y 289.602,Z 755.254,A -85,B 0,C 180,E1 -26900.22,E2 -26900.22} C_VEL
LIN {X 0,Y 292.187,Z 756.765,A -85,B 0,C 180,E1 -26901.702,E2 -26901.702} C_VEL
LIN {X 0,Y 294.345,Z 758.043,A -85,B 0,C 180,E1 -26903.144,E2 -26903.144} C_VEL
LIN {X 0,Y 296.408,Z 759.071,A -85,B 0,C 180,E1 -26904.764,E2 -26904.764} C_VEL
LIN {X 0,Y 297.666,Z 759.613,A -85,B 0,C 180,E1 -26905.938,E2 -26905.938} C_VEL
LIN {X 0,Y 298.756,Z 760.057,A -85,B 0,C 180,E1 -26907.303,E2 -26907.303} C_VEL
LIN {X 0,Y 299.406,Z 760.324,A -85,B 0,C 180,E1 -26908.655,E2 -26908.655} C_VEL
LIN {X 0,Y 299.739,Z 760.376,A -85,B 0,C 180,E1 -26910,E2 -26910} C_VEL
LIN {X 0,Y 299.404,Z 760.318,A -85,B 0,C 180,E1 -26911.345,E2 -26911.345} C_VEL
LIN {X 0,Y 298.757,Z 760.046,A -85,B 0,C 180,E1 -26912.697,E2 -26912.697} C_VEL
LIN {X 0,Y 297.672,Z 759.593,A -85,B 0,C 180,E1 -26914.062,E2 -26914.062} C_VEL
LIN {X 0,Y 296.165,Z 758.946,A -85,B 0,C 180,E1 -26915.447,E2 -26915.447} C_VEL
LIN {X 0,Y 294.34,Z 758.049,A -85,B 0,C 180,E1 -26916.856,E2 -26916.856} C_VEL
LIN {X 0,Y 291.505,Z 756.375,A -85,B 0,C 180,E1 -26918.71,E2 -26918.71} C_VEL
LIN {X 0,Y 288.284,Z 754.315,A -85,B 0,C 180,E1 -26920.535,E2 -26920.535} C_VEL
LIN {X 0,Y 283.237,Z 750.87,A -85,B 0,C 180,E1 -26922.904,E2 -26922.904} C_VEL
LIN {X 0,Y 278.658,Z 747.985,A -85,B 0,C 180,E1 -26924.608,E2 -26924.608} C_VEL
LIN {X 0,Y 271.824,Z 743.306,A -85,B 0,C 180,E1 -26926.939,E2 -26926.939} C_VEL
LIN {X 0,Y 263.561,Z 738.072,A -85,B 0,C 180,E1 -26929.398,E2 -26929.398} C_VEL
LIN {X 0,Y 254.111,Z 732.241,A -85,B 0,C 180,E1 -26932.104,E2 -26932.104} C_VEL
LIN {X 0,Y 244.171,Z 726.129,A -85,B 0,C 180,E1 -26934.953,E2 -26934.953} C_VEL
LIN {X 0,Y 227.514,Z 715.124,A -85,B 0,C 180,E1 -26940.127,E2 -26940.127} C_VEL
LIN {X 0,Y 216.628,Z 706.265,A -85,B 0,C 180,E1 -26944.141,E2 -26944.141} C_VEL
LIN {X 0,Y 207.6,Z 697.044,A -85,B 0,C 180,E1 -26948.086,E2 -26948.086} C_VEL
LIN {X 0,Y 199.396,Z 686.716,A -85,B 0,C 180,E1 -26952.255,E2 -26952.255} C_VEL
LIN {X 0,Y 193.65,Z 677.893,A -85,B 0,C 180,E1 -26955.606,E2 -26955.606} C_VEL
LIN {X 0,Y 188.155,Z 667.755,A -85,B 0,C 180,E1 -26959.183,E2 -26959.183} C_VEL
LIN {X 0,Y 183.329,Z 657.227,A -85,B 0,C 180,E1 -26962.6,E2 -26962.6} C_VEL
LIN {X 0,Y 178.743,Z 645.328,A -85,B 0,C 180,E1 -26966.065,E2 -26966.065} C_VEL
LIN {X 0,Y 172.056,Z 625.631,A -85,B 0,C 180,E1 -26971.34,E2 -26971.34} C_VEL
LIN {X 0,Y 168.774,Z 617.189,A -85,B 0,C 180,E1 -26974.273,E2 -26974.273} C_VEL
LIN {X 0,Y 165.401,Z 609.599,A -85,B 0,C 180,E1 -26977.682,E2 -26977.682} C_VEL
LIN {X 0,Y 162.362,Z 603.464,A -85,B 0,C 180,E1 -26981.312,E2 -26981.312} C_VEL
LIN {X 0,Y 160.41,Z 599.794,A -85,B 0,C 180,E1 -26984.109,E2 -26984.109} C_VEL
LIN {X 0,Y 158.946,Z 597.009,A -85,B 0,C 180,E1 -26986.643,E2 -26986.643} C_VEL
LIN {X 0,Y 157.365,Z 593.853,A -85,B 0,C 180,E1 -26990.198,E2 -26990.198} C_VEL
LIN {X 0,Y 155.708,Z 589.614,A -85,B 0,C 180,E1 -26998.708,E2 -26998.708} C_VEL
LIN {X 0,Y 155.704,Z 589.551,A -85,B 0,C 180,E1 -27000.648,E2 -27000.648} C_VEL
LIN {X 0,Y 155.897,Z 591.052,A -85,B 0,C 180,E1 -27003.879,E2 -27003.879} C_VEL
LIN {X 0,Y 157.576,Z 594.253,A -85,B 0,C 180,E1 -27009.953,E2 -27009.953} C_VEL
LIN {X 0,Y 159.656,Z 598.375,A -85,B 0,C 180,E1 -27014.256,E2 -27014.256} C_VEL
LIN {X 0,Y 161.693,Z 602.171,A -85,B 0,C 180,E1 -27017.388,E2 -27017.388} C_VEL
LIN {X 0,Y 164.216,Z 607.182,A -85,B 0,C 180,E1 -27020.595,E2 -27020.595} C_VEL
LIN {X 0,Y 165.54,Z 610.425,A -85,B 0,C 180,E1 -27022.136,E2 -27022.136} C_VEL
LIN {X 0,Y 168.128,Z 618.919,A -85,B 0,C 180,E1 -27025.04,E2 -27025.04} C_VEL
LIN {X 0,Y 164.959,Z 650.223,A -85,B 0,C 180,E1 -27026.009,E2 -27026.009} C_VEL
LIN {X 0,Y 162.22,Z 665.081,A -85,B 0,C 180,E1 -27026.671,E2 -27026.671} C_VEL
LIN {X 0,Y 158.132,Z 679.384,A -85,B 0,C 180,E1 -27027.616,E2 -27027.616} C_VEL
LIN {X 0,Y 154.116,Z 690.421,A -85,B 0,C 180,E1 -27028.62,E2 -27028.62} C_VEL
LIN {X 0,Y 149.839,Z 700.336,A -85,B 0,C 180,E1 -27029.808,E2 -27029.808} C_VEL
LIN {X 0,Y 144.927,Z 710.054,A -85,B 0,C 180,E1 -27031.276,E2 -27031.276} C_VEL
LIN {X 0,Y 139.435,Z 719.466,A -85,B 0,C 180,E1 -27033.077,E2 -27033.077} C_VEL
LIN {X 0,Y 134.025,Z 727.8,A -85,B 0,C 180,E1 -27035.145,E2 -27035.145} C_VEL
LIN {X 0,Y 128.482,Z 735.456,A -85,B 0,C 180,E1 -27037.52,E2 -27037.52} C_VEL
LIN {X 0,Y 122.392,Z 742.975,A -85,B 0,C 180,E1 -27040.463,E2 -27040.463} C_VEL
LIN {X 0,Y 116.614,Z 749.444,A -85,B 0,C 180,E1 -27043.682,E2 -27043.682} C_VEL
LIN {X 0,Y 110.356,Z 755.984,A -85,B 0,C 180,E1 -27048.035,E2 -27048.035} C_VEL
LIN {X 0,Y 104.811,Z 761.419,A -85,B 0,C 180,E1 -27052.881,E2 -27052.881} C_VEL
LIN {X 0,Y 100.118,Z 765.871,A -85,B 0,C 180,E1 -27058.233,E2 -27058.233} C_VEL
LIN {X 0,Y 96.317,Z 769.424,A -85,B 0,C 180,E1 -27064.037,E2 -27064.037} C_VEL
LIN {X 0,Y 94.241,Z 771.369,A -85,B 0,C 180,E1 -27068.108,E2 -27068.108} C_VEL
LIN {X 0,Y 91.687,Z 774.073,A -85,B 0,C 180,E1 -27076.706,E2 -27076.706} C_VEL
LIN {X 0,Y 90.837,Z 775.384,A -85,B 0,C 180,E1 -27085.563,E2 -27085.563} C_VEL
LIN {X 0,Y 90.975,Z 775.646,A -85,B 0,C 180,E1 -27090,E2 -27090} C_VEL
LIN {X 0,Y 91.078,Z 774.901,A -85,B 0,C 180,E1 -27098.878,E2 -27098.878} C_VEL
LIN {X 0,Y 91.687,Z 774.073,A -85,B 0,C 180,E1 -27103.294,E2 -27103.294} C_VEL
LIN {X 0,Y 94.24,Z 771.369,A -85,B 0,C 180,E1 -27111.893,E2 -27111.893} C_VEL
LIN {X 0,Y 98.73,Z 767.139,A -85,B 0,C 180,E1 -27119.886,E2 -27119.886} C_VEL
LIN {X 0,Y 102.957,Z 763.157,A -85,B 0,C 180,E1 -27125.226,E2 -27125.226} C_VEL
LIN {X 0,Y 108.423,Z 757.898,A -85,B 0,C 180,E1 -27130.405,E2 -27130.405} C_VEL
LIN {X 0,Y 114.483,Z 751.72,A -85,B 0,C 180,E1 -27134.907,E2 -27134.907} C_VEL
LIN {X 0,Y 120.038,Z 745.648,A -85,B 0,C 180,E1 -27138.286,E2 -27138.286} C_VEL
LIN {X 0,Y 126.028,Z 738.579,A -85,B 0,C 180,E1 -27141.324,E2 -27141.324} C_VEL
LIN {X 0,Y 131.822,Z 731.06,A -85,B 0,C 180,E1 -27143.852,E2 -27143.852} C_VEL
LIN {X 0,Y 138.119,Z 721.585,A -85,B 0,C 180,E1 -27146.429,E2 -27146.429} C_VEL
LIN {X 0,Y 143.551,Z 712.533,A -85,B 0,C 180,E1 -27148.28,E2 -27148.28} C_VEL
LIN {X 0,Y 148.402,Z 703.262,A -85,B 0,C 180,E1 -27149.799,E2 -27149.799} C_VEL
LIN {X 0,Y 152.677,Z 693.927,A -85,B 0,C 180,E1 -27150.996,E2 -27150.996} C_VEL
LIN {X 0,Y 156.681,Z 683.676,A -85,B 0,C 180,E1 -27152.015,E2 -27152.015} C_VEL
LIN {X 0,Y 160.114,Z 672.9,A -85,B 0,C 180,E1 -27152.849,E2 -27152.849} C_VEL
LIN {X 0,Y 163.008,Z 661.132,A -85,B 0,C 180,E1 -27153.529,E2 -27153.529} C_VEL
LIN {X 0,Y 165.004,Z 649.852,A -85,B 0,C 180,E1 -27153.982,E2 -27153.982} C_VEL
LIN {X 0,Y 168.131,Z 618.895,A -85,B 0,C 180,E1 -27154.96,E2 -27154.96} C_VEL
LIN {X 0,Y 165.355,Z 609.865,A -85,B 0,C 180,E1 -27158.084,E2 -27158.084} C_VEL
LIN {X 0,Y 163.785,Z 606.244,A -85,B 0,C 180,E1 -27159.922,E2 -27159.922} C_VEL
LIN {X 0,Y 161.065,Z 600.908,A -85,B 0,C 180,E1 -27163.522,E2 -27163.522} C_VEL
LIN {X 0,Y 159.723,Z 598.508,A -85,B 0,C 180,E1 -27165.628,E2 -27165.628} C_VEL
LIN {X 0,Y 158.936,Z 597.475,A -85,B 0,C 180,E1 -27166.961,E2 -27166.961} C_VEL
LIN {X 0,Y 158.131,Z 597.084,A -85,B 0,C 180,E1 -27168.349,E2 -27168.349} C_VEL
LIN {X 0,Y 156.644,Z 597.469,A -85,B 0,C 180,E1 -27171.196,E2 -27171.196} C_VEL
LIN {X 0,Y 155.498,Z 598.193,A -85,B 0,C 180,E1 -27174.124,E2 -27174.124} C_VEL
LIN {X 0,Y 154.996,Z 598.039,A -85,B 0,C 180,E1 -27176.338,E2 -27176.338} C_VEL
LIN {X 0,Y 154.914,Z 597.725,A -85,B 0,C 180,E1 -27177.069,E2 -27177.069} C_VEL
LIN {X 0,Y 154.841,Z 596.45,A -85,B 0,C 180,E1 -27179.999,E2 -27179.999} C_VEL
LIN {X 0,Y 154.852,Z 597.245,A -85,B 0,C 180,E1 -27182.356,E2 -27182.356} C_VEL
LIN {X 0,Y 156.474,Z 601.223,A -85,B 0,C 180,E1 -27189.859,E2 -27189.859} C_VEL
LIN {X 0,Y 158.362,Z 605.114,A -85,B 0,C 180,E1 -27194.018,E2 -27194.018} C_VEL
LIN {X 0,Y 160.463,Z 609.401,A -85,B 0,C 180,E1 -27197.441,E2 -27197.441} C_VEL
LIN {X 0,Y 163.242,Z 615.383,A -85,B 0,C 180,E1 -27201.082,E2 -27201.082} C_VEL
LIN {X 0,Y 166.254,Z 622.593,A -85,B 0,C 180,E1 -27204.408,E2 -27204.408} C_VEL
LIN {X 0,Y 169.05,Z 630.309,A -85,B 0,C 180,E1 -27207.153,E2 -27207.153} C_VEL
LIN {X 0,Y 171.997,Z 639.893,A -85,B 0,C 180,E1 -27209.849,E2 -27209.849} C_VEL
LIN {X 0,Y 176.07,Z 652.976,A -85,B 0,C 180,E1 -27213.541,E2 -27213.541} C_VEL
LIN {X 0,Y 180.21,Z 664.52,A -85,B 0,C 180,E1 -27217.19,E2 -27217.19} C_VEL
LIN {X 0,Y 184.892,Z 675.275,A -85,B 0,C 180,E1 -27220.971,E2 -27220.971} C_VEL
LIN {X 0,Y 190.037,Z 684.827,A -85,B 0,C 180,E1 -27224.639,E2 -27224.639} C_VEL
LIN {X 0,Y 196.542,Z 694.575,A -85,B 0,C 180,E1 -27228.669,E2 -27228.669} C_VEL
LIN {X 0,Y 205.631,Z 705.395,A -85,B 0,C 180,E1 -27233.446,E2 -27233.446} C_VEL
LIN {X 0,Y 215.798,Z 714.767,A -85,B 0,C 180,E1 -27237.858,E2 -27237.858} C_VEL
LIN {X 0,Y 229.411,Z 724.422,A -85,B 0,C 180,E1 -27242.672,E2 -27242.672} C_VEL
LIN {X 0,Y 241.56,Z 731.776,A -85,B 0,C 180,E1 -27246.41,E2 -27246.41} C_VEL
LIN {X 0,Y 254.14,Z 739.062,A -85,B 0,C 180,E1 -27250.089,E2 -27250.089} C_VEL
LIN {X 0,Y 263.632,Z 744.671,A -85,B 0,C 180,E1 -27252.948,E2 -27252.948} C_VEL
LIN {X 0,Y 269.485,Z 748.41,A -85,B 0,C 180,E1 -27254.883,E2 -27254.883} C_VEL
LIN {X 0,Y 274.573,Z 751.672,A -85,B 0,C 180,E1 -27256.682,E2 -27256.682} C_VEL
LIN {X 0,Y 278.703,Z 754.326,A -85,B 0,C 180,E1 -27258.362,E2 -27258.362} C_VEL
LIN {X 0,Y 281.932,Z 756.539,A -85,B 0,C 180,E1 -27259.951,E2 -27259.951} C_VEL
LIN {X 0,Y 284.65,Z 758.219,A -85,B 0,C 180,E1 -27261.481,E2 -27261.481} C_VEL
LIN {X 0,Y 286.987,Z 759.635,A -85,B 0,C 180,E1 -27262.967,E2 -27262.967} C_VEL
LIN {X 0,Y 289.371,Z 760.92,A -85,B 0,C 180,E1 -27264.721,E2 -27264.721} C_VEL
LIN {X 0,Y 290.62,Z 761.471,A -85,B 0,C 180,E1 -27265.84,E2 -27265.84} C_VEL
LIN {X 0,Y 291.801,Z 761.961,A -85,B 0,C 180,E1 -27267.239,E2 -27267.239} C_VEL
LIN {X 0,Y 292.538,Z 762.244,A -85,B 0,C 180,E1 -27268.623,E2 -27268.623} C_VEL
LIN {X 0,Y 292.902,Z 762.308,A -85,B 0,C 180,E1 -27270,E2 -27270} C_VEL
LIN {X 0,Y 292.537,Z 762.237,A -85,B 0,C 180,E1 -27271.377,E2 -27271.377} C_VEL
LIN {X 0,Y 291.802,Z 761.946,A -85,B 0,C 180,E1 -27272.761,E2 -27272.761} C_VEL
LIN {X 0,Y 290.624,Z 761.449,A -85,B 0,C 180,E1 -27274.16,E2 -27274.16} C_VEL
LIN {X 0,Y 288.984,Z 760.736,A -85,B 0,C 180,E1 -27275.582,E2 -27275.582} C_VEL
LIN {X 0,Y 286.997,Z 759.659,A -85,B 0,C 180,E1 -27277.033,E2 -27277.033} C_VEL
LIN {X 0,Y 284.366,Z 758.082,A -85,B 0,C 180,E1 -27278.672,E2 -27278.672} C_VEL
LIN {X 0,Y 281.958,Z 756.52,A -85,B 0,C 180,E1 -27280.048,E2 -27280.048} C_VEL
LIN {X 0,Y 278.731,Z 754.34,A -85,B 0,C 180,E1 -27281.637,E2 -27281.637} C_VEL
LIN {X 0,Y 274.488,Z 751.595,A -85,B 0,C 180,E1 -27283.36,E2 -27283.36} C_VEL
LIN {X 0,Y 266.879,Z 746.681,A -85,B 0,C 180,E1 -27286.018,E2 -27286.018} C_VEL
LIN {X 0,Y 262.508,Z 743.98,A -85,B 0,C 180,E1 -27287.405,E2 -27287.405} C_VEL
LIN {X 0,Y 251.598,Z 737.566,A -85,B 0,C 180,E1 -27290.65,E2 -27290.65} C_VEL
LIN {X 0,Y 239.212,Z 730.363,A -85,B 0,C 180,E1 -27294.287,E2 -27294.287} C_VEL
LIN {X 0,Y 224.723,Z 721.324,A -85,B 0,C 180,E1 -27298.877,E2 -27298.877} C_VEL
LIN {X 0,Y 213.68,Z 712.982,A -85,B 0,C 180,E1 -27302.999,E2 -27302.999} C_VEL
LIN {X 0,Y 202.785,Z 702.309,A -85,B 0,C 180,E1 -27307.961,E2 -27307.961} C_VEL
LIN {X 0,Y 193.227,Z 689.851,A -85,B 0,C 180,E1 -27313.33,E2 -27313.33} C_VEL
LIN {X 0,Y 186.311,Z 678.142,A -85,B 0,C 180,E1 -27317.968,E2 -27317.968} C_VEL
LIN {X 0,Y 181.507,Z 667.765,A -85,B 0,C 180,E1 -27321.72,E2 -27321.72} C_VEL
LIN {X 0,Y 177.112,Z 656.114,A -85,B 0,C 180,E1 -27325.508,E2 -27325.508} C_VEL
LIN {X 0,Y 173.489,Z 644.753,A -85,B 0,C 180,E1 -27328.828,E2 -27328.828} C_VEL
LIN {X 0,Y 169.182,Z 630.665,A -85,B 0,C 180,E1 -27332.727,E2 -27332.727} C_VEL
LIN {X 0,Y 166.489,Z 623.232,A -85,B 0,C 180,E1 -27335.348,E2 -27335.348} C_VEL
LIN {X 0,Y 163.844,Z 616.816,A -85,B 0,C 180,E1 -27338.205,E2 -27338.205} C_VEL
LIN {X 0,Y 161.268,Z 611.08,A -85,B 0,C 180,E1 -27341.427,E2 -27341.427} C_VEL
LIN {X 0,Y 159.034,Z 606.512,A -85,B 0,C 180,E1 -27344.789,E2 -27344.789} C_VEL
LIN {X 0,Y 157.691,Z 603.776,A -85,B 0,C 180,E1 -27347.283,E2 -27347.283} C_VEL
LIN {X 0,Y 156.189,Z 600.655,A -85,B 0,C 180,E1 -27350.94,E2 -27350.94} C_VEL
LIN {X 0,Y 154.839,Z 596.695,A -85,B 0,C 180,E1 -27358.701,E2 -27358.701} C_VEL
LIN {X 0,Y 154.843,Z 596.694,A -85,B 0,C 180,E1 -27360.976,E2 -27360.976} C_VEL
LIN {X 0,Y 156.443,Z 601.124,A -85,B 0,C 180,E1 -27369.373,E2 -27369.373} C_VEL
LIN {X 0,Y 158.277,Z 605.014,A -85,B 0,C 180,E1 -27373.482,E2 -27373.482} C_VEL
LIN {X 0,Y 160.298,Z 609.051,A -85,B 0,C 180,E1 -27376.805,E2 -27376.805} C_VEL
LIN {X 0,Y 162.871,Z 614.629,A -85,B 0,C 180,E1 -27380.252,E2 -27380.252} C_VEL
LIN {X 0,Y 164.955,Z 621.955,A -85,B 0,C 180,E1 -27382.922,E2 -27382.922} C_VEL
LIN {X 0,Y 161.953,Z 650.145,A -85,B 0,C 180,E1 -27383.753,E2 -27383.753} C_VEL
LIN {X 0,Y 159.071,Z 665.271,A -85,B 0,C 180,E1 -27384.408,E2 -27384.408} C_VEL
LIN {X 0,Y 154.972,Z 679.186,A -85,B 0,C 180,E1 -27385.291,E2 -27385.291} C_VEL
LIN {X 0,Y 150.84,Z 690.223,A -85,B 0,C 180,E1 -27386.249,E2 -27386.249} C_VEL
LIN {X 0,Y 146.432,Z 700.138,A -85,B 0,C 180,E1 -27387.392,E2 -27387.392} C_VEL
LIN {X 0,Y 141.368,Z 709.856,A -85,B 0,C 180,E1 -27388.813,E2 -27388.813} C_VEL
LIN {X 0,Y 135.67,Z 719.267,A -85,B 0,C 180,E1 -27390.549,E2 -27390.549} C_VEL
LIN {X 0,Y 129.77,Z 727.984,A -85,B 0,C 180,E1 -27392.684,E2 -27392.684} C_VEL
LIN {X 0,Y 124.276,Z 735.258,A -85,B 0,C 180,E1 -27394.917,E2 -27394.917} C_VEL
LIN {X 0,Y 117.895,Z 742.776,A -85,B 0,C 180,E1 -27397.829,E2 -27397.829} C_VEL
LIN {X 0,Y 111.802,Z 749.245,A -85,B 0,C 180,E1 -27401.034,E2 -27401.034} C_VEL
LIN {X 0,Y 105.143,Z 755.785,A -85,B 0,C 180,E1 -27405.426,E2 -27405.426} C_VEL
LIN {X 0,Y 99.203,Z 761.22,A -85,B 0,C 180,E1 -27410.388,E2 -27410.388} C_VEL
LIN {X 0,Y 94.102,Z 765.671,A -85,B 0,C 180,E1 -27415.936,E2 -27415.936} C_VEL
LIN {X 0,Y 89.948,Z 769.225,A -85,B 0,C 180,E1 -27422.044,E2 -27422.044} C_VEL
LIN {X 0,Y 87.658,Z 771.17,A -85,B 0,C 180,E1 -27426.368,E2 -27426.368} C_VEL
LIN {X 0,Y 84.756,Z 773.874,A -85,B 0,C 180,E1 -27435.596,E2 -27435.596} C_VEL
LIN {X 0,Y 83.759,Z 775.186,A -85,B 0,C 180,E1 -27445.187,E2 -27445.187} C_VEL
LIN {X 0,Y 83.881,Z 775.448,A -85,B 0,C 180,E1 -27450,E2 -27450} C_VEL
LIN {X 0,Y 84.039,Z 774.703,A -85,B 0,C 180,E1 -27459.628,E2 -27459.628} C_VEL
LIN {X 0,Y 84.756,Z 773.874,A -85,B 0,C 180,E1 -27464.404,E2 -27464.404} C_VEL
LIN {X 0,Y 87.656,Z 771.169,A -85,B 0,C 180,E1 -27473.633,E2 -27473.633} C_VEL
LIN {X 0,Y 92.6,Z 766.94,A -85,B 0,C 180,E1 -27482.091,E2 -27482.091} C_VEL
LIN {X 0,Y 97.202,Z 762.958,A -85,B 0,C 180,E1 -27487.658,E2 -27487.658} C_VEL
LIN {X 0,Y 103.071,Z 757.698,A -85,B 0,C 180,E1 -27492.988,E2 -27492.988} C_VEL
LIN {X 0,Y 109.521,Z 751.52,A -85,B 0,C 180,E1 -27497.556,E2 -27497.556} C_VEL
LIN {X 0,Y 115.42,Z 745.449,A -85,B 0,C 180,E1 -27500.926,E2 -27500.926} C_VEL
LIN {X 0,Y 121.69,Z 738.38,A -85,B 0,C 180,E1 -27503.952,E2 -27503.952} C_VEL
LIN {X 0,Y 127.98,Z 730.529,A -85,B 0,C 180,E1 -27506.537,E2 -27506.537} C_VEL
LIN {X 0,Y 133.616,Z 722.445,A -85,B 0,C 180,E1 -27508.727,E2 -27508.727} C_VEL
LIN {X 0,Y 139.24,Z 713.575,A -85,B 0,C 180,E1 -27510.535,E2 -27510.535} C_VEL
LIN {X 0,Y 144.232,Z 704.527,A -85,B 0,C 180,E1 -27512.025,E2 -27512.025} C_VEL
LIN {X 0,Y 149.367,Z 693.729,A -85,B 0,C 180,E1 -27513.376,E2 -27513.376} C_VEL
LIN {X 0,Y 153.486,Z 683.479,A -85,B 0,C 180,E1 -27514.349,E2 -27514.349} C_VEL
LIN {X 0,Y 156.901,Z 673.086,A -85,B 0,C 180,E1 -27515.127,E2 -27515.127} C_VEL
LIN {X 0,Y 159.929,Z 661.095,A -85,B 0,C 180,E1 -27515.804,E2 -27515.804} C_VEL
LIN {X 0,Y 162.023,Z 649.654,A -85,B 0,C 180,E1 -27516.233,E2 -27516.233} C_VEL
LIN {X 0,Y 164.932,Z 621.764,A -85,B 0,C 180,E1 -27517.117,E2 -27517.117} C_VEL
LIN {X 0,Y 162.77,Z 614.382,A -85,B 0,C 180,E1 -27519.874,E2 -27519.874} C_VEL
LIN {X 0,Y 160.35,Z 609.156,A -85,B 0,C 180,E1 -27523.119,E2 -27523.119} C_VEL
LIN {X 0,Y 158.712,Z 605.939,A -85,B 0,C 180,E1 -27525.723,E2 -27525.723} C_VEL
LIN {X 0,Y 157.487,Z 603.427,A -85,B 0,C 180,E1 -27528.088,E2 -27528.088} C_VEL
LIN {X 0,Y 156.223,Z 600.609,A -85,B 0,C 180,E1 -27531.266,E2 -27531.266} C_VEL
LIN {X 0,Y 154.914,Z 597.725,A -85,B 0,C 180,E1 -27537.069,E2 -27537.069} C_VEL
LIN {X 0,Y 154.778,Z 597.505,A -85,B 0,C 180,E1 -27538.503,E2 -27538.503} C_VEL
LIN {X 0,Y 154.564,Z 598.737,A -85,B 0,C 180,E1 -27540.635,E2 -27540.635} C_VEL
LIN {X 0,Y 154.417,Z 601.072,A -85,B 0,C 180,E1 -27542.675,E2 -27542.675} C_VEL
LIN {X 0,Y 154.458,Z 604.791,A -85,B 0,C 180,E1 -27545.424,E2 -27545.424} C_VEL
LIN {X 0,Y 154.822,Z 606.983,A -85,B 0,C 180,E1 -27547.554,E2 -27547.554} C_VEL
LIN {X 0,Y 155.034,Z 607.449,A -85,B 0,C 180,E1 -27548.289,E2 -27548.289} C_VEL
LIN {X 0,Y 155.57,Z 608.694,A -85,B 0,C 180,E1 -27549.916,E2 -27549.916} C_VEL
LIN {X 0,Y 157.018,Z 611.814,A -85,B 0,C 180,E1 -27553.26,E2 -27553.26} C_VEL
LIN {X 0,Y 158.889,Z 615.846,A -85,B 0,C 180,E1 -27556.553,E2 -27556.553} C_VEL
LIN {X 0,Y 161.499,Z 622.025,A -85,B 0,C 180,E1 -27560.257,E2 -27560.257} C_VEL
LIN {X 0,Y 164.006,Z 628.518,A -85,B 0,C 180,E1 -27563.255,E2 -27563.255} C_VEL
LIN {X 0,Y 166.651,Z 636.426,A -85,B 0,C 180,E1 -27566.08,E2 -27566.08} C_VEL
LIN {X 0,Y 170.861,Z 652.288,A -85,B 0,C 180,E1 -27570.656,E2 -27570.656} C_VEL
LIN {X 0,Y 173.934,Z 662.902,A -85,B 0,C 180,E1 -27574.009,E2 -27574.009} C_VEL
LIN {X 0,Y 177.474,Z 673.286,A -85,B 0,C 180,E1 -27577.629,E2 -27577.629} C_VEL
LIN {X 0,Y 182.072,Z 683.914,A -85,B 0,C 180,E1 -27581.746,E2 -27581.746} C_VEL
LIN {X 0,Y 188.048,Z 694.537,A -85,B 0,C 180,E1 -27586.261,E2 -27586.261} C_VEL
LIN {X 0,Y 195.188,Z 704.237,A -85,B 0,C 180,E1 -27590.725,E2 -27590.725} C_VEL
LIN {X 0,Y 202.535,Z 712.315,A -85,B 0,C 180,E1 -27594.63,E2 -27594.63} C_VEL
LIN {X 0,Y 212.858,Z 721.033,A -85,B 0,C 180,E1 -27599.141,E2 -27599.141} C_VEL
LIN {X 0,Y 224.947,Z 729.106,A -85,B 0,C 180,E1 -27603.507,E2 -27603.507} C_VEL
LIN {X 0,Y 237.085,Z 736.075,A -85,B 0,C 180,E1 -27607.334,E2 -27607.334} C_VEL
LIN {X 0,Y 246.556,Z 741.19,A -85,B 0,C 180,E1 -27610.159,E2 -27610.159} C_VEL
LIN {X 0,Y 256.82,Z 746.863,A -85,B 0,C 180,E1 -27613.29,E2 -27613.29} C_VEL
LIN {X 0,Y 263.695,Z 750.894,A -85,B 0,C 180,E1 -27615.593,E2 -27615.593} C_VEL
LIN {X 0,Y 270.244,Z 754.839,A -85,B 0,C 180,E1 -27617.992,E2 -27617.992} C_VEL
LIN {X 0,Y 273.912,Z 757.243,A -85,B 0,C 180,E1 -27619.654,E2 -27619.654} C_VEL
LIN {X 0,Y 277.188,Z 759.397,A -85,B 0,C 180,E1 -27621.422,E2 -27621.422} C_VEL
LIN {X 0,Y 279.435,Z 760.813,A -85,B 0,C 180,E1 -27622.776,E2 -27622.776} C_VEL
LIN {X 0,Y 282.287,Z 762.275,A -85,B 0,C 180,E1 -27624.778,E2 -27624.778} C_VEL
LIN {X 0,Y 283.381,Z 762.789,A -85,B 0,C 180,E1 -27625.733,E2 -27625.733} C_VEL
LIN {X 0,Y 284.7,Z 763.368,A -85,B 0,C 180,E1 -27627.17,E2 -27627.17} C_VEL
LIN {X 0,Y 285.548,Z 763.688,A -85,B 0,C 180,E1 -27628.59,E2 -27628.59} C_VEL
LIN {X 0,Y 285.957,Z 763.771,A -85,B 0,C 180,E1 -27630,E2 -27630} C_VEL
LIN {X 0,Y 285.547,Z 763.679,A -85,B 0,C 180,E1 -27631.41,E2 -27631.41} C_VEL
LIN {X 0,Y 284.702,Z 763.348,A -85,B 0,C 180,E1 -27632.83,E2 -27632.83} C_VEL
LIN {X 0,Y 283.401,Z 762.779,A -85,B 0,C 180,E1 -27634.266,E2 -27634.266} C_VEL
LIN {X 0,Y 281.601,Z 761.973,A -85,B 0,C 180,E1 -27635.729,E2 -27635.729} C_VEL
LIN {X 0,Y 279.437,Z 760.82,A -85,B 0,C 180,E1 -27637.224,E2 -27637.224} C_VEL
LIN {X 0,Y 276.898,Z 759.196,A -85,B 0,C 180,E1 -27638.759,E2 -27638.759} C_VEL
LIN {X 0,Y 272.222,Z 756.069,A -85,B 0,C 180,E1 -27641.176,E2 -27641.176} C_VEL
LIN {X 0,Y 270.3,Z 754.837,A -85,B 0,C 180,E1 -27642.005,E2 -27642.005} C_VEL
LIN {X 0,Y 263.7,Z 750.896,A -85,B 0,C 180,E1 -27644.407,E2 -27644.407} C_VEL
LIN {X 0,Y 256.832,Z 746.84,A -85,B 0,C 180,E1 -27646.719,E2 -27646.719} C_VEL
LIN {X 0,Y 245.792,Z 740.787,A -85,B 0,C 180,E1 -27650.067,E2 -27650.067} C_VEL
LIN {X 0,Y 234.955,Z 734.819,A -85,B 0,C 180,E1 -27653.342,E2 -27653.342} C_VEL
LIN {X 0,Y 217.947,Z 724.689,A -85,B 0,C 180,E1 -27658.926,E2 -27658.926} C_VEL
LIN {X 0,Y 206.571,Z 716.022,A -85,B 0,C 180,E1 -27663.496,E2 -27663.496} C_VEL
LIN {X 0,Y 196.931,Z 706.382,A -85,B 0,C 180,E1 -27668.269,E2 -27668.269} C_VEL
LIN {X 0,Y 190.153,Z 697.636,A -85,B 0,C 180,E1 -27672.339,E2 -27672.339} C_VEL
LIN {X 0,Y 184.412,Z 688.366,A -85,B 0,C 180,E1 -27676.392,E2 -27676.392} C_VEL
LIN {X 0,Y 179.565,Z 678.466,A -85,B 0,C 180,E1 -27680.405,E2 -27680.405} C_VEL
LIN {X 0,Y 175.92,Z 669.063,A -85,B 0,C 180,E1 -27683.897,E2 -27683.897} C_VEL
LIN {X 0,Y 172.161,Z 657.201,A -85,B 0,C 180,E1 -27687.855,E2 -27687.855} C_VEL
LIN {X 0,Y 168.866,Z 644.683,A -85,B 0,C 180,E1 -27691.565,E2 -27691.565} C_VEL
LIN {X 0,Y 166.22,Z 635.05,A -85,B 0,C 180,E1 -27694.362,E2 -27694.362} C_VEL
LIN {X 0,Y 163.631,Z 627.459,A -85,B 0,C 180,E1 -27697.174,E2 -27697.174} C_VEL
LIN {X 0,Y 160.939,Z 620.671,A -85,B 0,C 180,E1 -27700.473,E2 -27700.473} C_VEL
LIN {X 0,Y 158.587,Z 615.243,A -85,B 0,C 180,E1 -27703.921,E2 -27703.921} C_VEL
LIN {X 0,Y 156.565,Z 610.701,A -85,B 0,C 180,E1 -27707.71,E2 -27707.71} C_VEL
LIN {X 0,Y 155.096,Z 607.502,A -85,B 0,C 180,E1 -27711.533,E2 -27711.533} C_VEL
LIN {X 0,Y 153.961,Z 603.653,A -85,B 0,C 180,E1 -27719.347,E2 -27719.347} C_VEL
LIN {X 0,Y 153.966,Z 603.832,A -85,B 0,C 180,E1 -27720.982,E2 -27720.982} C_VEL
LIN {X 0,Y 155.328,Z 607.985,A -85,B 0,C 180,E1 -27728.785,E2 -27728.785} C_VEL
LIN {X 0,Y 157.006,Z 611.825,A -85,B 0,C 180,E1 -27732.852,E2 -27732.852} C_VEL
LIN {X 0,Y 158.702,Z 615.439,A -85,B 0,C 180,E1 -27735.863,E2 -27735.863} C_VEL
LIN {X 0,Y 160.816,Z 620.435,A -85,B 0,C 180,E1 -27738.978,E2 -27738.978} C_VEL
LIN {X 0,Y 161.985,Z 624.943,A -85,B 0,C 180,E1 -27740.689,E2 -27740.689} C_VEL
LIN {X 0,Y 159.226,Z 649.957,A -85,B 0,C 180,E1 -27741.415,E2 -27741.415} C_VEL
LIN {X 0,Y 156.293,Z 664.982,A -85,B 0,C 180,E1 -27742.033,E2 -27742.033} C_VEL
LIN {X 0,Y 152.076,Z 678.988,A -85,B 0,C 180,E1 -27742.874,E2 -27742.874} C_VEL
LIN {X 0,Y 147.842,Z 690.025,A -85,B 0,C 180,E1 -27743.784,E2 -27743.784} C_VEL
LIN {X 0,Y 143.305,Z 699.94,A -85,B 0,C 180,E1 -27744.87,E2 -27744.87} C_VEL
LIN {X 0,Y 138.08,Z 709.657,A -85,B 0,C 180,E1 -27746.226,E2 -27746.226} C_VEL
LIN {X 0,Y 132.187,Z 719.068,A -85,B 0,C 180,E1 -27747.886,E2 -27747.886} C_VEL
LIN {X 0,Y 126.321,Z 727.45,A -85,B 0,C 180,E1 -27749.865,E2 -27749.865} C_VEL
LIN {X 0,Y 120.345,Z 735.06,A -85,B 0,C 180,E1 -27752.139,E2 -27752.139} C_VEL
LIN {X 0,Y 113.67,Z 742.578,A -85,B 0,C 180,E1 -27754.995,E2 -27754.995} C_VEL
LIN {X 0,Y 107.247,Z 749.045,A -85,B 0,C 180,E1 -27758.154,E2 -27758.154} C_VEL
LIN {X 0,Y 100.183,Z 755.585,A -85,B 0,C 180,E1 -27762.559,E2 -27762.559} C_VEL
LIN {X 0,Y 93.791,Z 761.02,A -85,B 0,C 180,E1 -27767.594,E2 -27767.594} C_VEL
LIN {X 0,Y 88.195,Z 765.511,A -85,B 0,C 180,E1 -27773.388,E2 -27773.388} C_VEL
LIN {X 0,Y 83.676,Z 769.024,A -85,B 0,C 180,E1 -27779.739,E2 -27779.739} C_VEL
LIN {X 0,Y 81.173,Z 770.971,A -85,B 0,C 180,E1 -27784.349,E2 -27784.349} C_VEL
LIN {X 0,Y 77.87,Z 773.675,A -85,B 0,C 180,E1 -27794.291,E2 -27794.291} C_VEL
LIN {X 0,Y 76.663,Z 774.988,A -85,B 0,C 180,E1 -27804.74,E2 -27804.74} C_VEL
LIN {X 0,Y 76.778,Z 775.25,A -85,B 0,C 180,E1 -27810,E2 -27810} C_VEL
LIN {X 0,Y 77.009,Z 774.503,A -85,B 0,C 180,E1 -27820.517,E2 -27820.517} C_VEL
LIN {X 0,Y 77.87,Z 773.675,A -85,B 0,C 180,E1 -27825.709,E2 -27825.709} C_VEL
LIN {X 0,Y 81.171,Z 770.971,A -85,B 0,C 180,E1 -27835.652,E2 -27835.652} C_VEL
LIN {X 0,Y 86.626,Z 766.74,A -85,B 0,C 180,E1 -27844.604,E2 -27844.604} C_VEL
LIN {X 0,Y 91.835,Z 762.6,A -85,B 0,C 180,E1 -27850.577,E2 -27850.577} C_VEL
LIN {X 0,Y 97.963,Z 757.499,A -85,B 0,C 180,E1 -27855.84,E2 -27855.84} C_VEL
LIN {X 0,Y 104.825,Z 751.321,A -85,B 0,C 180,E1 -27860.444,E2 -27860.444} C_VEL
LIN {X 0,Y 111.06,Z 745.25,A -85,B 0,C 180,E1 -27863.786,E2 -27863.786} C_VEL
LIN {X 0,Y 117.631,Z 738.181,A -85,B 0,C 180,E1 -27866.765,E2 -27866.765} C_VEL
LIN {X 0,Y 123.618,Z 731.084,A -85,B 0,C 180,E1 -27869.069,E2 -27869.069} C_VEL
LIN {X 0,Y 130.071,Z 722.247,A -85,B 0,C 180,E1 -27871.402,E2 -27871.402} C_VEL
LIN {X 0,Y 135.882,Z 713.377,A -85,B 0,C 180,E1 -27873.148,E2 -27873.148} C_VEL
LIN {X 0,Y 141.038,Z 704.329,A -85,B 0,C 180,E1 -27874.576,E2 -27874.576} C_VEL
LIN {X 0,Y 146.316,Z 693.531,A -85,B 0,C 180,E1 -27875.868,E2 -27875.868} C_VEL
LIN {X 0,Y 150.537,Z 683.28,A -85,B 0,C 180,E1 -27876.797,E2 -27876.797} C_VEL
LIN {X 0,Y 154.23,Z 672.253,A -85,B 0,C 180,E1 -27877.561,E2 -27877.561} C_VEL
LIN {X 0,Y 157.125,Z 661.042,A -85,B 0,C 180,E1 -27878.156,E2 -27878.156} C_VEL
LIN {X 0,Y 159.251,Z 649.751,A -85,B 0,C 180,E1 -27878.563,E2 -27878.563} C_VEL
LIN {X 0,Y 162.007,Z 625.014,A -85,B 0,C 180,E1 -27879.281,E2 -27879.281} C_VEL
LIN {X 0,Y 160.642,Z 619.954,A -85,B 0,C 180,E1 -27881.267,E2 -27881.267} C_VEL
LIN {X 0,Y 158.44,Z 614.86,A -85,B 0,C 180,E1 -27884.564,E2 -27884.564} C_VEL
LIN {X 0,Y 156.304,Z 610.233,A -85,B 0,C 180,E1 -27888.662,E2 -27888.662} C_VEL
LIN {X 0,Y 155.125,Z 607.479,A -85,B 0,C 180,E1 -27891.86,E2 -27891.86} C_VEL
LIN {X 0,Y 153.973,Z 603.522,A -85,B 0,C 180,E1 -27899.999,E2 -27899.999} C_VEL
LIN {X 0,Y 153.97,Z 604.438,A -85,B 0,C 180,E1 -27902.37,E2 -27902.37} C_VEL
LIN {X 0,Y 155.034,Z 607.449,A -85,B 0,C 180,E1 -27908.289,E2 -27908.289} C_VEL
LIN {X 0,Y 155.687,Z 609.34,A -85,B 0,C 180,E1 -27910.332,E2 -27910.332} C_VEL
LIN {X 0,Y 156.29,Z 612.415,A -85,B 0,C 180,E1 -27912.187,E2 -27912.187} C_VEL
LIN {X 0,Y 158.651,Z 625.609,A -85,B 0,C 180,E1 -27917.754,E2 -27917.754} C_VEL
LIN {X 0,Y 161.117,Z 632.303,A -85,B 0,C 180,E1 -27921.174,E2 -27921.174} C_VEL
LIN {X 0,Y 163.404,Z 639.473,A -85,B 0,C 180,E1 -27923.956,E2 -27923.956} C_VEL
LIN {X 0,Y 165.592,Z 648.869,A -85,B 0,C 180,E1 -27926.82,E2 -27926.82} C_VEL
LIN {X 0,Y 168.387,Z 661.5,A -85,B 0,C 180,E1 -27930.748,E2 -27930.748} C_VEL
LIN {X 0,Y 171.57,Z 673.556,A -85,B 0,C 180,E1 -27934.992,E2 -27934.992} C_VEL
LIN {X 0,Y 175.817,Z 685.516,A -85,B 0,C 180,E1 -27939.758,E2 -27939.758} C_VEL
LIN {X 0,Y 180.904,Z 695.937,A -85,B 0,C 180,E1 -27944.368,E2 -27944.368} C_VEL
LIN {X 0,Y 186.874,Z 705.102,A -85,B 0,C 180,E1 -27948.776,E2 -27948.776} C_VEL
LIN {X 0,Y 193.672,Z 713.334,A -85,B 0,C 180,E1 -27952.97,E2 -27952.97} C_VEL
LIN {X 0,Y 202.7,Z 721.739,A -85,B 0,C 180,E1 -27957.533,E2 -27957.533} C_VEL
LIN {X 0,Y 214.367,Z 729.962,A -85,B 0,C 180,E1 -27962.273,E2 -27962.273} C_VEL
LIN {X 0,Y 228.81,Z 738.13,A -85,B 0,C 180,E1 -27967.138,E2 -27967.138} C_VEL
LIN {X 0,Y 238.937,Z 743.34,A -85,B 0,C 180,E1 -27970.257,E2 -27970.257} C_VEL
LIN {X 0,Y 246.676,Z 747.274,A -85,B 0,C 180,E1 -27972.635,E2 -27972.635} C_VEL
LIN {X 0,Y 254.477,Z 751.346,A -85,B 0,C 180,E1 -27975.148,E2 -27975.148} C_VEL
LIN {X 0,Y 261.277,Z 755.095,A -85,B 0,C 180,E1 -27977.574,E2 -27977.574} C_VEL
LIN {X 0,Y 265.659,Z 757.553,A -85,B 0,C 180,E1 -27979.328,E2 -27979.328} C_VEL
LIN {X 0,Y 269.98,Z 760.317,A -85,B 0,C 180,E1 -27981.565,E2 -27981.565} C_VEL
LIN {X 0,Y 271.706,Z 761.39,A -85,B 0,C 180,E1 -27982.569,E2 -27982.569} C_VEL
LIN {X 0,Y 275.174,Z 763.245,A -85,B 0,C 180,E1 -27984.906,E2 -27984.906} C_VEL
LIN {X 0,Y 277.508,Z 764.388,A -85,B 0,C 180,E1 -27987.097,E2 -27987.097} C_VEL
LIN {X 0,Y 278.469,Z 764.782,A -85,B 0,C 180,E1 -27988.554,E2 -27988.554} C_VEL
LIN {X 0,Y 278.942,Z 764.883,A -85,B 0,C 180,E1 -27990,E2 -27990} C_VEL
LIN {X 0,Y 278.469,Z 764.769,A -85,B 0,C 180,E1 -27991.446,E2 -27991.446} C_VEL
LIN {X 0,Y 277.514,Z 764.369,A -85,B 0,C 180,E1 -27992.903,E2 -27992.903} C_VEL
LIN {X 0,Y 275.175,Z 763.231,A -85,B 0,C 180,E1 -27995.096,E2 -27995.096} C_VEL
LIN {X 0,Y 271.691,Z 761.391,A -85,B 0,C 180,E1 -27997.431,E2 -27997.431} C_VEL
LIN {X 0,Y 267.414,Z 758.625,A -85,B 0,C 180,E1 -27999.836,E2 -27999.836} C_VEL
LIN {X 0,Y 264.905,Z 757.091,A -85,B 0,C 180,E1 -28001.007,E2 -28001.007} C_VEL
LIN {X 0,Y 259.68,Z 754.181,A -85,B 0,C 180,E1 -28003.021,E2 -28003.021} C_VEL
LIN {X 0,Y 251.897,Z 749.945,A -85,B 0,C 180,E1 -28005.734,E2 -28005.734} C_VEL
LIN {X 0,Y 242.787,Z 745.286,A -85,B 0,C 180,E1 -28008.567,E2 -28008.567} C_VEL
LIN {X 0,Y 231.339,Z 739.407,A -85,B 0,C 180,E1 -28012.095,E2 -28012.095} C_VEL
LIN {X 0,Y 216.162,Z 731.07,A -85,B 0,C 180,E1 -28017.076,E2 -28017.076} C_VEL
LIN {X 0,Y 204.097,Z 722.863,A -85,B 0,C 180,E1 -28021.835,E2 -28021.835} C_VEL
LIN {X 0,Y 193.666,Z 713.347,A -85,B 0,C 180,E1 -28027.028,E2 -28027.028} C_VEL
LIN {X 0,Y 185.327,Z 702.914,A -85,B 0,C 180,E1 -28032.315,E2 -28032.315} C_VEL
LIN {X 0,Y 178.941,Z 692.19,A -85,B 0,C 180,E1 -28037.353,E2 -28037.353} C_VEL
LIN {X 0,Y 173.867,Z 680.422,A -85,B 0,C 180,E1 -28042.348,E2 -28042.348} C_VEL
LIN {X 0,Y 170.639,Z 670.23,A -85,B 0,C 180,E1 -28046.221,E2 -28046.221} C_VEL
LIN {X 0,Y 167.592,Z 658.274,A -85,B 0,C 180,E1 -28050.293,E2 -28050.293} C_VEL
LIN {X 0,Y 164.864,Z 645.473,A -85,B 0,C 180,E1 -28054.176,E2 -28054.176} C_VEL
LIN {X 0,Y 163.038,Z 638.259,A -85,B 0,C 180,E1 -28056.473,E2 -28056.473} C_VEL
LIN {X 0,Y 160.767,Z 631.284,A -85,B 0,C 180,E1 -28059.28,E2 -28059.28} C_VEL
LIN {X 0,Y 158.283,Z 624.691,A -85,B 0,C 180,E1 -28062.811,E2 -28062.811} C_VEL
LIN {X 0,Y 156.276,Z 619.772,A -85,B 0,C 180,E1 -28066.333,E2 -28066.333} C_VEL
LIN {X 0,Y 155.01,Z 616.874,A -85,B 0,C 180,E1 -28069.138,E2 -28069.138} C_VEL
LIN {X 0,Y 154.018,Z 614.371,A -85,B 0,C 180,E1 -28072.133,E2 -28072.133} C_VEL
LIN {X 0,Y 153.092,Z 610.729,A -85,B 0,C 180,E1 -28079.344,E2 -28079.344} C_VEL
LIN {X 0,Y 153.092,Z 610.886,A -85,B 0,C 180,E1 -28080.823,E2 -28080.823} C_VEL
LIN {X 0,Y 154.236,Z 614.829,A -85,B 0,C 180,E1 -28088.198,E2 -28088.198} C_VEL
LIN {X 0,Y 155.605,Z 618.274,A -85,B 0,C 180,E1 -28091.881,E2 -28091.881} C_VEL
LIN {X 0,Y 157.363,Z 622.348,A -85,B 0,C 180,E1 -28095.276,E2 -28095.276} C_VEL
LIN {X 0,Y 158.914,Z 626.488,A -85,B 0,C 180,E1 -28097.785,E2 -28097.785} C_VEL
LIN {X 0,Y 159.274,Z 628.101,A -85,B 0,C 180,E1 -28098.405,E2 -28098.405} C_VEL
LIN {X 0,Y 156.595,Z 650.983,A -85,B 0,C 180,E1 -28099.039,E2 -28099.039} C_VEL
LIN {X 0,Y 153.172,Z 666.86,A -85,B 0,C 180,E1 -28099.674,E2 -28099.674} C_VEL
LIN {X 0,Y 149.464,Z 678.791,A -85,B 0,C 180,E1 -28100.37,E2 -28100.37} C_VEL
LIN {X 0,Y 145.119,Z 689.827,A -85,B 0,C 180,E1 -28101.213,E2 -28101.213} C_VEL
LIN {X 0,Y 140.462,Z 699.742,A -85,B 0,C 180,E1 -28102.238,E2 -28102.238} C_VEL
LIN {X 0,Y 135.085,Z 709.459,A -85,B 0,C 180,E1 -28103.516,E2 -28103.516} C_VEL
LIN {X 0,Y 129.021,Z 718.87,A -85,B 0,C 180,E1 -28105.099,E2 -28105.099} C_VEL
LIN {X 0,Y 122.418,Z 727.891,A -85,B 0,C 180,E1 -28107.151,E2 -28107.151} C_VEL
LIN {X 0,Y 116.645,Z 734.938,A -85,B 0,C 180,E1 -28109.205,E2 -28109.205} C_VEL
LIN {X 0,Y 109.745,Z 742.38,A -85,B 0,C 180,E1 -28111.951,E2 -28111.951} C_VEL
LIN {X 0,Y 102.993,Z 748.846,A -85,B 0,C 180,E1 -28115.032,E2 -28115.032} C_VEL
LIN {X 0,Y 95.507,Z 755.387,A -85,B 0,C 180,E1 -28119.409,E2 -28119.409} C_VEL
LIN {X 0,Y 88.646,Z 760.821,A -85,B 0,C 180,E1 -28124.478,E2 -28124.478} C_VEL
LIN {X 0,Y 83.006,Z 764.994,A -85,B 0,C 180,E1 -28129.892,E2 -28129.892} C_VEL
LIN {X 0,Y 77.566,Z 768.824,A -85,B 0,C 180,E1 -28137.069,E2 -28137.069} C_VEL
LIN {X 0,Y 74.807,Z 770.772,A -85,B 0,C 180,E1 -28141.983,E2 -28141.983} C_VEL
LIN {X 0,Y 71.006,Z 773.475,A -85,B 0,C 180,E1 -28152.727,E2 -28152.727} C_VEL
LIN {X 0,Y 69.576,Z 774.789,A -85,B 0,C 180,E1 -28164.203,E2 -28164.203} C_VEL
LIN {X 0,Y 69.673,Z 775.052,A -85,B 0,C 180,E1 -28170,E2 -28170} C_VEL
LIN {X 0,Y 70.014,Z 774.305,A -85,B 0,C 180,E1 -28181.581,E2 -28181.581} C_VEL
LIN {X 0,Y 71.006,Z 773.475,A -85,B 0,C 180,E1 -28187.273,E2 -28187.273} C_VEL
LIN {X 0,Y 74.805,Z 770.772,A -85,B 0,C 180,E1 -28198.018,E2 -28198.018} C_VEL
LIN {X 0,Y 80.821,Z 766.54,A -85,B 0,C 180,E1 -28207.495,E2 -28207.495} C_VEL
LIN {X 0,Y 86.532,Z 762.401,A -85,B 0,C 180,E1 -28213.657,E2 -28213.657} C_VEL
LIN {X 0,Y 93.134,Z 757.3,A -85,B 0,C 180,E1 -28218.99,E2 -28218.99} C_VEL
LIN {X 0,Y 100.415,Z 751.121,A -85,B 0,C 180,E1 -28223.597,E2 -28223.597} C_VEL
LIN {X 0,Y 106.998,Z 745.051,A -85,B 0,C 180,E1 -28226.871,E2 -28226.871} C_VEL
LIN {X 0,Y 113.882,Z 737.982,A -85,B 0,C 180,E1 -28229.764,E2 -28229.764} C_VEL
LIN {X 0,Y 119.596,Z 731.527,A -85,B 0,C 180,E1 -28231.817,E2 -28231.817} C_VEL
LIN {X 0,Y 126.809,Z 722.048,A -85,B 0,C 180,E1 -28234.235,E2 -28234.235} C_VEL
LIN {X 0,Y 132.828,Z 713.179,A -85,B 0,C 180,E1 -28235.88,E2 -28235.88} C_VEL
LIN {X 0,Y 138.138,Z 704.131,A -85,B 0,C 180,E1 -28237.238,E2 -28237.238} C_VEL
LIN {X 0,Y 143.554,Z 693.332,A -85,B 0,C 180,E1 -28238.46,E2 -28238.46} C_VEL
LIN {X 0,Y 147.881,Z 683.082,A -85,B 0,C 180,E1 -28239.328,E2 -28239.328} C_VEL
LIN {X 0,Y 151.518,Z 672.545,A -85,B 0,C 180,E1 -28240.016,E2 -28240.016} C_VEL
LIN {X 0,Y 154.717,Z 660.398,A -85,B 0,C 180,E1 -28240.62,E2 -28240.62} C_VEL
LIN {X 0,Y 156.693,Z 650.259,A -85,B 0,C 180,E1 -28240.96,E2 -28240.96} C_VEL
LIN {X 0,Y 159.274,Z 628.047,A -85,B 0,C 180,E1 -28241.602,E2 -28241.602} C_VEL
LIN {X 0,Y 158.505,Z 625.214,A -85,B 0,C 180,E1 -28242.864,E2 -28242.864} C_VEL
LIN {X 0,Y 156.477,Z 620.213,A -85,B 0,C 180,E1 -28246.338,E2 -28246.338} C_VEL
LIN {X 0,Y 154.879,Z 616.562,A -85,B 0,C 180,E1 -28249.871,E2 -28249.871} C_VEL
LIN {X 0,Y 153.948,Z 614.183,A -85,B 0,C 180,E1 -28252.787,E2 -28252.787} C_VEL
LIN {X 0,Y 153.105,Z 610.587,A -85,B 0,C 180,E1 -28259.999,E2 -28259.999} C_VEL
LIN {X 0,Y 153.296,Z 612.778,A -85,B 0,C 180,E1 -28264.642,E2 -28264.642} C_VEL
LIN {X 0,Y 154.257,Z 614.94,A -85,B 0,C 180,E1 -28268.679,E2 -28268.679} C_VEL
LIN {X 0,Y 155.696,Z 618.461,A -85,B 0,C 180,E1 -28272.47,E2 -28272.47} C_VEL
LIN {X 0,Y 157.429,Z 622.521,A -85,B 0,C 180,E1 -28275.784,E2 -28275.784} C_VEL
LIN {X 0,Y 158.651,Z 625.609,A -85,B 0,C 180,E1 -28277.754,E2 -28277.754} C_VEL
LIN {X 0,Y 159.541,Z 629.685,A -85,B 0,C 180,E1 -28279.271,E2 -28279.271} C_VEL
LIN {X 0,Y 160.584,Z 637.784,A -85,B 0,C 180,E1 -28281.302,E2 -28281.302} C_VEL
LIN {X 0,Y 161.6,Z 647.891,A -85,B 0,C 180,E1 -28283.623,E2 -28283.623} C_VEL
LIN {X 0,Y 162.047,Z 650.959,A -85,B 0,C 180,E1 -28284.526,E2 -28284.526} C_VEL
LIN {X 0,Y 163.922,Z 662.294,A -85,B 0,C 180,E1 -28288.138,E2 -28288.138} C_VEL
LIN {X 0,Y 166.194,Z 673.815,A -85,B 0,C 180,E1 -28292.249,E2 -28292.249} C_VEL
LIN {X 0,Y 168.927,Z 684.092,A -85,B 0,C 180,E1 -28296.358,E2 -28296.358} C_VEL
LIN {X 0,Y 172.493,Z 693.848,A -85,B 0,C 180,E1 -28300.683,E2 -28300.683} C_VEL
LIN {X 0,Y 177.462,Z 703.638,A -85,B 0,C 180,E1 -28305.466,E2 -28305.466} C_VEL
LIN {X 0,Y 183.414,Z 712.264,A -85,B 0,C 180,E1 -28310.026,E2 -28310.026} C_VEL
LIN {X 0,Y 192.168,Z 721.689,A -85,B 0,C 180,E1 -28315.371,E2 -28315.371} C_VEL
LIN {X 0,Y 200.216,Z 728.285,A -85,B 0,C 180,E1 -28319.314,E2 -28319.314} C_VEL
LIN {X 0,Y 213.969,Z 736.766,A -85,B 0,C 180,E1 -28324.724,E2 -28324.724} C_VEL
LIN {X 0,Y 226.175,Z 742.976,A -85,B 0,C 180,E1 -28328.777,E2 -28328.777} C_VEL
LIN {X 0,Y 236.472,Z 747.852,A -85,B 0,C 180,E1 -28331.995,E2 -28331.995} C_VEL
LIN {X 0,Y 244.019,Z 751.397,A -85,B 0,C 180,E1 -28334.367,E2 -28334.367} C_VEL
LIN {X 0,Y 249.502,Z 754.054,A -85,B 0,C 180,E1 -28336.205,E2 -28336.205} C_VEL
LIN {X 0,Y 256.981,Z 757.799,A -85,B 0,C 180,E1 -28338.964,E2 -28338.964} C_VEL
LIN {X 0,Y 260.829,Z 759.885,A -85,B 0,C 180,E1 -28340.696,E2 -28340.696} C_VEL
LIN {X 0,Y 263.825,Z 761.642,A -85,B 0,C 180,E1 -28342.346,E2 -28342.346} C_VEL
LIN {X 0,Y 268.047,Z 763.879,A -85,B 0,C 180,E1 -28345.082,E2 -28345.082} C_VEL
LIN {X 0,Y 270.199,Z 764.908,A -85,B 0,C 180,E1 -28347.018,E2 -28347.018} C_VEL
LIN {X 0,Y 271.291,Z 765.317,A -85,B 0,C 180,E1 -28348.516,E2 -28348.516} C_VEL
LIN {X 0,Y 271.866,Z 765.434,A -85,B 0,C 180,E1 -28350,E2 -28350} C_VEL
LIN {X 0,Y 271.293,Z 765.316,A -85,B 0,C 180,E1 -28351.484,E2 -28351.484} C_VEL
LIN {X 0,Y 270.208,Z 764.908,A -85,B 0,C 180,E1 -28352.982,E2 -28352.982} C_VEL
LIN {X 0,Y 268.048,Z 763.876,A -85,B 0,C 180,E1 -28354.922,E2 -28354.922} C_VEL
LIN {X 0,Y 263.837,Z 761.642,A -85,B 0,C 180,E1 -28357.654,E2 -28357.654} C_VEL
LIN {X 0,Y 260.887,Z 759.884,A -85,B 0,C 180,E1 -28359.301,E2 -28359.301} C_VEL
LIN {X 0,Y 256.91,Z 757.802,A -85,B 0,C 180,E1 -28361.04,E2 -28361.04} C_VEL
LIN {X 0,Y 252.051,Z 755.358,A -85,B 0,C 180,E1 -28362.889,E2 -28362.889} C_VEL
LIN {X 0,Y 246.406,Z 752.522,A -85,B 0,C 180,E1 -28364.874,E2 -28364.874} C_VEL
LIN {X 0,Y 236.471,Z 747.854,A -85,B 0,C 180,E1 -28368.004,E2 -28368.004} C_VEL
LIN {X 0,Y 226.196,Z 742.939,A -85,B 0,C 180,E1 -28371.237,E2 -28371.237} C_VEL
LIN {X 0,Y 211.444,Z 735.39,A -85,B 0,C 180,E1 -28376.181,E2 -28376.181} C_VEL
LIN {X 0,Y 198.129,Z 726.711,A -85,B 0,C 180,E1 -28381.646,E2 -28381.646} C_VEL
LIN {X 0,Y 187.256,Z 716.794,A -85,B 0,C 180,E1 -28387.461,E2 -28387.461} C_VEL
LIN {X 0,Y 179.198,Z 706.418,A -85,B 0,C 180,E1 -28393.082,E2 -28393.082} C_VEL
LIN {X 0,Y 174.329,Z 697.786,A -85,B 0,C 180,E1 -28397.411,E2 -28397.411} C_VEL
LIN {X 0,Y 170.344,Z 688.398,A -85,B 0,C 180,E1 -28401.768,E2 -28401.768} C_VEL
LIN {X 0,Y 167.315,Z 678.587,A -85,B 0,C 180,E1 -28405.898,E2 -28405.898} C_VEL
LIN {X 0,Y 165.253,Z 669.637,A -85,B 0,C 180,E1 -28409.315,E2 -28409.315} C_VEL
LIN {X 0,Y 163.027,Z 657.512,A -85,B 0,C 180,E1 -28413.432,E2 -28413.432} C_VEL
LIN {X 0,Y 161.04,Z 645.604,A -85,B 0,C 180,E1 -28417.166,E2 -28417.166} C_VEL
LIN {X 0,Y 159.142,Z 638.43,A -85,B 0,C 180,E1 -28419.953,E2 -28419.953} C_VEL
LIN {X 0,Y 156.991,Z 631.978,A -85,B 0,C 180,E1 -28423.241,E2 -28423.241} C_VEL
LIN {X 0,Y 155.097,Z 626.784,A -85,B 0,C 180,E1 -28426.793,E2 -28426.793} C_VEL
LIN {X 0,Y 153.713,Z 623.363,A -85,B 0,C 180,E1 -28430.15,E2 -28430.15} C_VEL
LIN {X 0,Y 152.915,Z 621.143,A -85,B 0,C 180,E1 -28432.906,E2 -28432.906} C_VEL
LIN {X 0,Y 152.232,Z 617.702,A -85,B 0,C 180,E1 -28440.001,E2 -28440.001} C_VEL
LIN {X 0,Y 153.109,Z 621.548,A -85,B 0,C 180,E1 -28447.419,E2 -28447.419} C_VEL
LIN {X 0,Y 154.36,Z 625.055,A -85,B 0,C 180,E1 -28451.179,E2 -28451.179} C_VEL
LIN {X 0,Y 155.68,Z 628.336,A -85,B 0,C 180,E1 -28454.001,E2 -28454.001} C_VEL
LIN {X 0,Y 156.782,Z 631.419,A -85,B 0,C 180,E1 -28456.017,E2 -28456.017} C_VEL
LIN {X 0,Y 154.307,Z 651.582,A -85,B 0,C 180,E1 -28456.575,E2 -28456.575} C_VEL
LIN {X 0,Y 151.113,Z 666.066,A -85,B 0,C 180,E1 -28457.112,E2 -28457.112} C_VEL
LIN {X 0,Y 147.139,Z 678.592,A -85,B 0,C 180,E1 -28457.772,E2 -28457.772} C_VEL
LIN {X 0,Y 142.703,Z 689.629,A -85,B 0,C 180,E1 -28458.554,E2 -28458.554} C_VEL
LIN {X 0,Y 137.931,Z 699.543,A -85,B 0,C 180,E1 -28459.505,E2 -28459.505} C_VEL
LIN {X 0,Y 132.404,Z 709.26,A -85,B 0,C 180,E1 -28460.688,E2 -28460.688} C_VEL
LIN {X 0,Y 126.158,Z 718.671,A -85,B 0,C 180,E1 -28462.162,E2 -28462.162} C_VEL
LIN {X 0,Y 119.338,Z 727.689,A -85,B 0,C 180,E1 -28464.105,E2 -28464.105} C_VEL
LIN {X 0,Y 113.038,Z 735.058,A -85,B 0,C 180,E1 -28466.161,E2 -28466.161} C_VEL
LIN {X 0,Y 106.143,Z 742.181,A -85,B 0,C 180,E1 -28468.682,E2 -28468.682} C_VEL
LIN {X 0,Y 97.71,Z 749.785,A -85,B 0,C 180,E1 -28472.315,E2 -28472.315} C_VEL
LIN {X 0,Y 91.138,Z 755.187,A -85,B 0,C 180,E1 -28475.935,E2 -28475.935} C_VEL
LIN {X 0,Y 83.778,Z 760.621,A -85,B 0,C 180,E1 -28480.977,E2 -28480.977} C_VEL
LIN {X 0,Y 78.204,Z 764.477,A -85,B 0,C 180,E1 -28485.97,E2 -28485.97} C_VEL
LIN {X 0,Y 71.659,Z 768.625,A -85,B 0,C 180,E1 -28493.954,E2 -28493.954} C_VEL
LIN {X 0,Y 68.568,Z 770.572,A -85,B 0,C 180,E1 -28499.171,E2 -28499.171} C_VEL
LIN {X 0,Y 64.209,Z 773.276,A -85,B 0,C 180,E1 -28510.831,E2 -28510.831} C_VEL
LIN {X 0,Y 62.514,Z 774.591,A -85,B 0,C 180,E1 -28523.545,E2 -28523.545} C_VEL
LIN {X 0,Y 62.563,Z 774.853,A -85,B 0,C 180,E1 -28530,E2 -28530} C_VEL
LIN {X 0,Y 63.059,Z 774.106,A -85,B 0,C 180,E1 -28542.879,E2 -28542.879} C_VEL
LIN {X 0,Y 64.209,Z 773.276,A -85,B 0,C 180,E1 -28549.169,E2 -28549.169} C_VEL
LIN {X 0,Y 68.566,Z 770.572,A -85,B 0,C 180,E1 -28560.83,E2 -28560.83} C_VEL
LIN {X 0,Y 75.258,Z 766.34,A -85,B 0,C 180,E1 -28570.82,E2 -28570.82} C_VEL
LIN {X 0,Y 81.513,Z 762.202,A -85,B 0,C 180,E1 -28577.126,E2 -28577.126} C_VEL
LIN {X 0,Y 88.606,Z 757.1,A -85,B 0,C 180,E1 -28582.482,E2 -28582.482} C_VEL
LIN {X 0,Y 96.35,Z 750.922,A -85,B 0,C 180,E1 -28587.016,E2 -28587.016} C_VEL
LIN {X 0,Y 103.278,Z 744.853,A -85,B 0,C 180,E1 -28590.182,E2 -28590.182} C_VEL
LIN {X 0,Y 110.471,Z 737.784,A -85,B 0,C 180,E1 -28592.954,E2 -28592.954} C_VEL
LIN {X 0,Y 117.049,Z 730.511,A -85,B 0,C 180,E1 -28595.145,E2 -28595.145} C_VEL
LIN {X 0,Y 123.882,Z 721.85,A -85,B 0,C 180,E1 -28597.2,E2 -28597.2} C_VEL
LIN {X 0,Y 130.081,Z 712.98,A -85,B 0,C 180,E1 -28598.742,E2 -28598.742} C_VEL
LIN {X 0,Y 135.544,Z 703.933,A -85,B 0,C 180,E1 -28600.012,E2 -28600.012} C_VEL
LIN {X 0,Y 141.099,Z 693.134,A -85,B 0,C 180,E1 -28601.147,E2 -28601.147} C_VEL
LIN {X 0,Y 145.523,Z 682.883,A -85,B 0,C 180,E1 -28601.949,E2 -28601.949} C_VEL
LIN {X 0,Y 149.075,Z 672.919,A -85,B 0,C 180,E1 -28602.544,E2 -28602.544} C_VEL
LIN {X 0,Y 152.379,Z 660.786,A -85,B 0,C 180,E1 -28603.115,E2 -28603.115} C_VEL
LIN {X 0,Y 154.608,Z 649.529,A -85,B 0,C 180,E1 -28603.455,E2 -28603.455} C_VEL
LIN {X 0,Y 156.785,Z 631.347,A -85,B 0,C 180,E1 -28603.991,E2 -28603.991} C_VEL
LIN {X 0,Y 155.073,Z 626.72,A -85,B 0,C 180,E1 -28607.238,E2 -28607.238} C_VEL
LIN {X 0,Y 153.723,Z 623.356,A -85,B 0,C 180,E1 -28610.521,E2 -28610.521} C_VEL
LIN {X 0,Y 152.879,Z 620.961,A -85,B 0,C 180,E1 -28613.482,E2 -28613.482} C_VEL
LIN {X 0,Y 152.236,Z 617.669,A -85,B 0,C 180,E1 -28619.999,E2 -28619.999} C_VEL
LIN {X 0,Y 153.174,Z 621.8,A -85,B 0,C 180,E1 -28628.076,E2 -28628.076} C_VEL
LIN {X 0,Y 154.447,Z 625.212,A -85,B 0,C 180,E1 -28631.766,E2 -28631.766} C_VEL
LIN {X 0,Y 156.004,Z 629.216,A -85,B 0,C 180,E1 -28635.012,E2 -28635.012} C_VEL
LIN {X 0,Y 158.127,Z 635.273,A -85,B 0,C 180,E1 -28638.561,E2 -28638.561} C_VEL
LIN {X 0,Y 160.194,Z 642.213,A -85,B 0,C 180,E1 -28641.619,E2 -28641.619} C_VEL
LIN {X 0,Y 161.883,Z 649.945,A -85,B 0,C 180,E1 -28644.217,E2 -28644.217} C_VEL
LIN {X 0,Y 162.047,Z 650.959,A -85,B 0,C 180,E1 -28644.526,E2 -28644.526} C_VEL
LIN {X 0,Y 162.471,Z 655.673,A -85,B 0,C 180,E1 -28645.777,E2 -28645.777} C_VEL
LIN {X 0,Y 161.66,Z 671.284,A -85,B 0,C 180,E1 -28648.821,E2 -28648.821} C_VEL
LIN {X 0,Y 161.595,Z 675.896,A -85,B 0,C 180,E1 -28650.11,E2 -28650.11} C_VEL
LIN {X 0,Y 161.764,Z 677.238,A -85,B 0,C 180,E1 -28650.61,E2 -28650.61} C_VEL
LIN {X 0,Y 163.405,Z 685.45,A -85,B 0,C 180,E1 -28653.994,E2 -28653.994} C_VEL
LIN {X 0,Y 166.341,Z 695.562,A -85,B 0,C 180,E1 -28658.647,E2 -28658.647} C_VEL
LIN {X 0,Y 170.54,Z 705.371,A -85,B 0,C 180,E1 -28663.65,E2 -28663.65} C_VEL
LIN {X 0,Y 175.913,Z 714.069,A -85,B 0,C 180,E1 -28668.51,E2 -28668.51} C_VEL
LIN {X 0,Y 183.181,Z 722.691,A -85,B 0,C 180,E1 -28673.675,E2 -28673.675} C_VEL
LIN {X 0,Y 191.727,Z 730.147,A -85,B 0,C 180,E1 -28678.442,E2 -28678.442} C_VEL
LIN {X 0,Y 203.808,Z 737.881,A -85,B 0,C 180,E1 -28683.708,E2 -28683.708} C_VEL
LIN {X 0,Y 218.48,Z 745.174,A -85,B 0,C 180,E1 -28688.883,E2 -28688.883} C_VEL
LIN {X 0,Y 228.842,Z 749.711,A -85,B 0,C 180,E1 -28692.181,E2 -28692.181} C_VEL
LIN {X 0,Y 236.021,Z 752.819,A -85,B 0,C 180,E1 -28694.455,E2 -28694.455} C_VEL
LIN {X 0,Y 242.446,Z 755.634,A -85,B 0,C 180,E1 -28696.591,E2 -28696.591} C_VEL
LIN {X 0,Y 250.214,Z 759.058,A -85,B 0,C 180,E1 -28699.439,E2 -28699.439} C_VEL
LIN {X 0,Y 252.382,Z 760.122,A -85,B 0,C 180,E1 -28700.382,E2 -28700.382} C_VEL
LIN {X 0,Y 255.836,Z 761.868,A -85,B 0,C 180,E1 -28702.105,E2 -28702.105} C_VEL
LIN {X 0,Y 258.582,Z 763.278,A -85,B 0,C 180,E1 -28703.759,E2 -28703.759} C_VEL
LIN {X 0,Y 261.042,Z 764.355,A -85,B 0,C 180,E1 -28705.367,E2 -28705.367} C_VEL
LIN {X 0,Y 262.85,Z 765.124,A -85,B 0,C 180,E1 -28706.935,E2 -28706.935} C_VEL
LIN {X 0,Y 264.08,Z 765.577,A -85,B 0,C 180,E1 -28708.475,E2 -28708.475} C_VEL
LIN {X 0,Y 264.754,Z 765.724,A -85,B 0,C 180,E1 -28710,E2 -28710} C_VEL
LIN {X 0,Y 264.083,Z 765.577,A -85,B 0,C 180,E1 -28711.525,E2 -28711.525} C_VEL
LIN {X 0,Y 262.858,Z 765.125,A -85,B 0,C 180,E1 -28713.065,E2 -28713.065} C_VEL
LIN {X 0,Y 260.914,Z 764.316,A -85,B 0,C 180,E1 -28714.714,E2 -28714.714} C_VEL
LIN {X 0,Y 258.586,Z 763.277,A -85,B 0,C 180,E1 -28716.241,E2 -28716.241} C_VEL
LIN {X 0,Y 255.544,Z 761.695,A -85,B 0,C 180,E1 -28718.086,E2 -28718.086} C_VEL
LIN {X 0,Y 252.383,Z 760.122,A -85,B 0,C 180,E1 -28719.618,E2 -28719.618} C_VEL
LIN {X 0,Y 247.889,Z 758.057,A -85,B 0,C 180,E1 -28721.447,E2 -28721.447} C_VEL
LIN {X 0,Y 242.504,Z 755.632,A -85,B 0,C 180,E1 -28723.406,E2 -28723.406} C_VEL
LIN {X 0,Y 234.124,Z 752.001,A -85,B 0,C 180,E1 -28726.144,E2 -28726.144} C_VEL
LIN {X 0,Y 223.634,Z 747.438,A -85,B 0,C 180,E1 -28729.478,E2 -28729.478} C_VEL
LIN {X 0,Y 208.569,Z 740.416,A -85,B 0,C 180,E1 -28734.525,E2 -28734.525} C_VEL
LIN {X 0,Y 193.936,Z 731.77,A -85,B 0,C 180,E1 -28740.486,E2 -28740.486} C_VEL
LIN {X 0,Y 185.265,Z 724.682,A -85,B 0,C 180,E1 -28745.078,E2 -28745.078} C_VEL
LIN {X 0,Y 177.258,Z 715.872,A -85,B 0,C 180,E1 -28750.436,E2 -28750.436} C_VEL
LIN {X 0,Y 172.09,Z 708.164,A -85,B 0,C 180,E1 -28754.833,E2 -28754.833} C_VEL
LIN {X 0,Y 167.241,Z 698.012,A -85,B 0,C 180,E1 -28760.145,E2 -28760.145} C_VEL
LIN {X 0,Y 164.367,Z 689.212,A -85,B 0,C 180,E1 -28764.33,E2 -28764.33} C_VEL
LIN {X 0,Y 162.305,Z 680.15,A -85,B 0,C 180,E1 -28768.236,E2 -28768.236} C_VEL
LIN {X 0,Y 160.469,Z 668.73,A -85,B 0,C 180,E1 -28772.623,E2 -28772.623} C_VEL
LIN {X 0,Y 159.201,Z 657.969,A -85,B 0,C 180,E1 -28776.288,E2 -28776.288} C_VEL
LIN {X 0,Y 158.177,Z 649.535,A -85,B 0,C 180,E1 -28779.096,E2 -28779.096} C_VEL
LIN {X 0,Y 156.71,Z 642.944,A -85,B 0,C 180,E1 -28781.821,E2 -28781.821} C_VEL
LIN {X 0,Y 154.887,Z 636.798,A -85,B 0,C 180,E1 -28785.205,E2 -28785.205} C_VEL
LIN {X 0,Y 153.354,Z 632.355,A -85,B 0,C 180,E1 -28788.599,E2 -28788.599} C_VEL
LIN {X 0,Y 152.456,Z 629.779,A -85,B 0,C 180,E1 -28791.218,E2 -28791.218} C_VEL
LIN {X 0,Y 151.84,Z 627.916,A -85,B 0,C 180,E1 -28793.69,E2 -28793.69} C_VEL
LIN {X 0,Y 151.355,Z 624.845,A -85,B 0,C 180,E1 -28800.001,E2 -28800.001} C_VEL
LIN {X 0,Y 152.073,Z 628.491,A -85,B 0,C 180,E1 -28806.907,E2 -28806.907} C_VEL
LIN {X 0,Y 153.124,Z 631.741,A -85,B 0,C 180,E1 -28810.413,E2 -28810.413} C_VEL
LIN {X 0,Y 154.439,Z 635.415,A -85,B 0,C 180,E1 -28813.488,E2 -28813.488} C_VEL
LIN {X 0,Y 154.423,Z 636.415,A -85,B 0,C 180,E1 -28813.654,E2 -28813.654} C_VEL
LIN {X 0,Y 151.936,Z 654.171,A -85,B 0,C 180,E1 -28814.104,E2 -28814.104} C_VEL
LIN {X 0,Y 148.65,Z 667.617,A -85,B 0,C 180,E1 -28814.587,E2 -28814.587} C_VEL
LIN {X 0,Y 144.715,Z 679.467,A -85,B 0,C 180,E1 -28815.162,E2 -28815.162} C_VEL
LIN {X 0,Y 140.608,Z 689.431,A -85,B 0,C 180,E1 -28815.815,E2 -28815.815} C_VEL
LIN {X 0,Y 135.719,Z 699.345,A -85,B 0,C 180,E1 -28816.67,E2 -28816.67} C_VEL
LIN {X 0,Y 130.057,Z 709.061,A -85,B 0,C 180,E1 -28817.75,E2 -28817.75} C_VEL
LIN {X 0,Y 123.651,Z 718.472,A -85,B 0,C 180,E1 -28819.109,E2 -28819.109} C_VEL
LIN {X 0,Y 116.601,Z 727.49,A -85,B 0,C 180,E1 -28820.897,E2 -28820.897} C_VEL
LIN {X 0,Y 109.772,Z 735.179,A -85,B 0,C 180,E1 -28822.928,E2 -28822.928} C_VEL
LIN {X 0,Y 102.911,Z 741.982,A -85,B 0,C 180,E1 -28825.197,E2 -28825.197} C_VEL
LIN {X 0,Y 95.534,Z 748.449,A -85,B 0,C 180,E1 -28828.022,E2 -28828.022} C_VEL
LIN {X 0,Y 87.129,Z 754.988,A -85,B 0,C 180,E1 -28832.121,E2 -28832.121} C_VEL
LIN {X 0,Y 79.279,Z 760.422,A -85,B 0,C 180,E1 -28837.077,E2 -28837.077} C_VEL
LIN {X 0,Y 72.645,Z 764.604,A -85,B 0,C 180,E1 -28842.629,E2 -28842.629} C_VEL
LIN {X 0,Y 66.008,Z 768.425,A -85,B 0,C 180,E1 -28850.296,E2 -28850.296} C_VEL
LIN {X 0,Y 62.532,Z 770.372,A -85,B 0,C 180,E1 -28855.81,E2 -28855.81} C_VEL
LIN {X 0,Y 57.509,Z 773.077,A -85,B 0,C 180,E1 -28868.493,E2 -28868.493} C_VEL
LIN {X 0,Y 55.451,Z 774.393,A -85,B 0,C 180,E1 -28882.719,E2 -28882.719} C_VEL
LIN {X 0,Y 55.474,Z 774.656,A -85,B 0,C 180,E1 -28890,E2 -28890} C_VEL
LIN {X 0,Y 56.118,Z 773.907,A -85,B 0,C 180,E1 -28904.505,E2 -28904.505} C_VEL
LIN {X 0,Y 57.509,Z 773.077,A -85,B 0,C 180,E1 -28911.507,E2 -28911.507} C_VEL
LIN {X 0,Y 62.529,Z 770.372,A -85,B 0,C 180,E1 -28924.192,E2 -28924.192} C_VEL
LIN {X 0,Y 67.956,Z 767.406,A -85,B 0,C 180,E1 -28932.238,E2 -28932.238} C_VEL
LIN {X 0,Y 74.44,Z 763.571,A -85,B 0,C 180,E1 -28939.049,E2 -28939.049} C_VEL
LIN {X 0,Y 81.818,Z 758.805,A -85,B 0,C 180,E1 -28944.688,E2 -28944.688} C_VEL
LIN {X 0,Y 91.246,Z 751.86,A -85,B 0,C 180,E1 -28950.052,E2 -28950.052} C_VEL
LIN {X 0,Y 99.929,Z 744.654,A -85,B 0,C 180,E1 -28953.725,E2 -28953.725} C_VEL
LIN {X 0,Y 107.425,Z 737.586,A -85,B 0,C 180,E1 -28956.333,E2 -28956.333} C_VEL
LIN {X 0,Y 113.54,Z 731.128,A -85,B 0,C 180,E1 -28958.197,E2 -28958.197} C_VEL
LIN {X 0,Y 121.299,Z 721.651,A -85,B 0,C 180,E1 -28960.304,E2 -28960.304} C_VEL
LIN {X 0,Y 127.671,Z 712.781,A -85,B 0,C 180,E1 -28961.723,E2 -28961.723} C_VEL
LIN {X 0,Y 133.284,Z 703.735,A -85,B 0,C 180,E1 -28962.882,E2 -28962.882} C_VEL
LIN {X 0,Y 138.965,Z 692.936,A -85,B 0,C 180,E1 -28963.92,E2 -28963.92} C_VEL
LIN {X 0,Y 143.481,Z 682.685,A -85,B 0,C 180,E1 -28964.646,E2 -28964.646} C_VEL
LIN {X 0,Y 147.362,Z 671.852,A -85,B 0,C 180,E1 -28965.226,E2 -28965.226} C_VEL
LIN {X 0,Y 150.397,Z 660.93,A -85,B 0,C 180,E1 -28965.685,E2 -28965.685} C_VEL
LIN {X 0,Y 152.737,Z 649.331,A -85,B 0,C 180,E1 -28966.011,E2 -28966.011} C_VEL
LIN {X 0,Y 154.478,Z 635.559,A -85,B 0,C 180,E1 -28966.426,E2 -28966.426} C_VEL
LIN {X 0,Y 153.227,Z 632.031,A -85,B 0,C 180,E1 -28969.313,E2 -28969.313} C_VEL
LIN {X 0,Y 152.395,Z 629.616,A -85,B 0,C 180,E1 -28971.817,E2 -28971.817} C_VEL
LIN {X 0,Y 151.872,Z 627.843,A -85,B 0,C 180,E1 -28974.001,E2 -28974.001} C_VEL
LIN {X 0,Y 151.354,Z 624.849,A -85,B 0,C 180,E1 -28979.999,E2 -28979.999} C_VEL
LIN {X 0,Y 152.128,Z 628.724,A -85,B 0,C 180,E1 -28987.548,E2 -28987.548} C_VEL
LIN {X 0,Y 153.195,Z 631.909,A -85,B 0,C 180,E1 -28990.986,E2 -28990.986} C_VEL
LIN {X 0,Y 154.41,Z 635.358,A -85,B 0,C 180,E1 -28993.825,E2 -28993.825} C_VEL
LIN {X 0,Y 156.249,Z 641.289,A -85,B 0,C 180,E1 -28997.362,E2 -28997.362} C_VEL
LIN {X 0,Y 157.782,Z 647.738,A -85,B 0,C 180,E1 -29000.227,E2 -29000.227} C_VEL
LIN {X 0,Y 158.797,Z 654.231,A -85,B 0,C 180,E1 -29002.525,E2 -29002.525} C_VEL
LIN {X 0,Y 159.785,Z 663.042,A -85,B 0,C 180,E1 -29005.364,E2 -29005.364} C_VEL
LIN {X 0,Y 161.249,Z 674.074,A -85,B 0,C 180,E1 -29009.346,E2 -29009.346} C_VEL
LIN {X 0,Y 161.764,Z 677.238,A -85,B 0,C 180,E1 -29010.61,E2 -29010.61} C_VEL
LIN {X 0,Y 162.225,Z 681.441,A -85,B 0,C 180,E1 -29012.077,E2 -29012.077} C_VEL
LIN {X 0,Y 161.624,Z 689.209,A -85,B 0,C 180,E1 -29014.251,E2 -29014.251} C_VEL
LIN {X 0,Y 160.993,Z 696.706,A -85,B 0,C 180,E1 -29016.524,E2 -29016.524} C_VEL
LIN {X 0,Y 161.43,Z 700.487,A -85,B 0,C 180,E1 -29018.112,E2 -29018.112} C_VEL
LIN {X 0,Y 166.475,Z 712.34,A -85,B 0,C 180,E1 -29024.715,E2 -29024.715} C_VEL
LIN {X 0,Y 172.882,Z 721.733,A -85,B 0,C 180,E1 -29030.567,E2 -29030.567} C_VEL
LIN {X 0,Y 179.608,Z 728.793,A -85,B 0,C 180,E1 -29035.255,E2 -29035.255} C_VEL
LIN {X 0,Y 189.238,Z 736.257,A -85,B 0,C 180,E1 -29040.54,E2 -29040.54} C_VEL
LIN {X 0,Y 203.284,Z 743.899,A -85,B 0,C 180,E1 -29046.369,E2 -29046.369} C_VEL
LIN {X 0,Y 215.914,Z 749.419,A -85,B 0,C 180,E1 -29050.723,E2 -29050.723} C_VEL
LIN {X 0,Y 226.518,Z 753.632,A -85,B 0,C 180,E1 -29054.111,E2 -29054.111} C_VEL
LIN {X 0,Y 232.368,Z 755.923,A -85,B 0,C 180,E1 -29055.998,E2 -29055.998} C_VEL
LIN {X 0,Y 238.442,Z 758.322,A -85,B 0,C 180,E1 -29058.093,E2 -29058.093} C_VEL
LIN {X 0,Y 243.651,Z 760.366,A -85,B 0,C 180,E1 -29060.034,E2 -29060.034} C_VEL
LIN {X 0,Y 248.285,Z 762.377,A -85,B 0,C 180,E1 -29062.179,E2 -29062.179} C_VEL
LIN {X 0,Y 250.723,Z 763.498,A -85,B 0,C 180,E1 -29063.562,E2 -29063.562} C_VEL
LIN {X 0,Y 253.779,Z 764.708,A -85,B 0,C 180,E1 -29065.52,E2 -29065.52} C_VEL
LIN {X 0,Y 255.42,Z 765.332,A -85,B 0,C 180,E1 -29066.845,E2 -29066.845} C_VEL
LIN {X 0,Y 256.827,Z 765.776,A -85,B 0,C 180,E1 -29068.432,E2 -29068.432} C_VEL
LIN {X 0,Y 257.641,Z 765.922,A -85,B 0,C 180,E1 -29070,E2 -29070} C_VEL
LIN {X 0,Y 256.831,Z 765.776,A -85,B 0,C 180,E1 -29071.568,E2 -29071.568} C_VEL
LIN {X 0,Y 255.431,Z 765.333,A -85,B 0,C 180,E1 -29073.154,E2 -29073.154} C_VEL
LIN {X 0,Y 253.351,Z 764.57,A -85,B 0,C 180,E1 -29074.774,E2 -29074.774} C_VEL
LIN {X 0,Y 250.743,Z 763.498,A -85,B 0,C 180,E1 -29076.437,E2 -29076.437} C_VEL
LIN {X 0,Y 247.646,Z 762.101,A -85,B 0,C 180,E1 -29078.157,E2 -29078.157} C_VEL
LIN {X 0,Y 242.84,Z 760.077,A -85,B 0,C 180,E1 -29080.272,E2 -29080.272} C_VEL
LIN {X 0,Y 237.373,Z 757.863,A -85,B 0,C 180,E1 -29082.305,E2 -29082.305} C_VEL
LIN {X 0,Y 229.214,Z 754.667,A -85,B 0,C 180,E1 -29085.025,E2 -29085.025} C_VEL
LIN {X 0,Y 221.188,Z 751.531,A -85,B 0,C 180,E1 -29087.599,E2 -29087.599} C_VEL
LIN {X 0,Y 208.599,Z 746.307,A -85,B 0,C 180,E1 -29091.752,E2 -29091.752} C_VEL
LIN {X 0,Y 193.87,Z 739.056,A -85,B 0,C 180,E1 -29097.361,E2 -29097.361} C_VEL
LIN {X 0,Y 183.349,Z 731.973,A -85,B 0,C 180,E1 -29102.514,E2 -29102.514} C_VEL
LIN {X 0,Y 174.683,Z 723.888,A -85,B 0,C 180,E1 -29108.028,E2 -29108.028} C_VEL
LIN {X 0,Y 168.027,Z 714.971,A -85,B 0,C 180,E1 -29113.669,E2 -29113.669} C_VEL
LIN {X 0,Y 163.936,Z 707.079,A -85,B 0,C 180,E1 -29118.273,E2 -29118.273} C_VEL
LIN {X 0,Y 161.127,Z 699.557,A -85,B 0,C 180,E1 -29122.365,E2 -29122.365} C_VEL
LIN {X 0,Y 158.705,Z 689.483,A -85,B 0,C 180,E1 -29127.285,E2 -29127.285} C_VEL
LIN {X 0,Y 157.391,Z 680.223,A -85,B 0,C 180,E1 -29131.315,E2 -29131.315} C_VEL
LIN {X 0,Y 156.397,Z 668.653,A -85,B 0,C 180,E1 -29135.758,E2 -29135.758} C_VEL
LIN {X 0,Y 155.767,Z 657.772,A -85,B 0,C 180,E1 -29139.468,E2 -29139.468} C_VEL
LIN {X 0,Y 154.967,Z 650.571,A -85,B 0,C 180,E1 -29142.287,E2 -29142.287} C_VEL
LIN {X 0,Y 153.696,Z 644.681,A -85,B 0,C 180,E1 -29145.311,E2 -29145.311} C_VEL
LIN {X 0,Y 152.324,Z 639.593,A -85,B 0,C 180,E1 -29148.838,E2 -29148.838} C_VEL
LIN {X 0,Y 151.327,Z 636.497,A -85,B 0,C 180,E1 -29151.992,E2 -29151.992} C_VEL
LIN {X 0,Y 150.828,Z 634.748,A -85,B 0,C 180,E1 -29154.319,E2 -29154.319} C_VEL
LIN {X 0,Y 150.469,Z 632.059,A -85,B 0,C 180,E1 -29160.001,E2 -29160.001} C_VEL
LIN {X 0,Y 151.026,Z 635.32,A -85,B 0,C 180,E1 -29166.263,E2 -29166.263} C_VEL
LIN {X 0,Y 151.941,Z 638.5,A -85,B 0,C 180,E1 -29169.706,E2 -29169.706} C_VEL
LIN {X 0,Y 152.45,Z 640.01,A -85,B 0,C 180,E1 -29171.11,E2 -29171.11} C_VEL
LIN {X 0,Y 150.107,Z 655.086,A -85,B 0,C 180,E1 -29171.512,E2 -29171.512} C_VEL
LIN {X 0,Y 147.026,Z 667.42,A -85,B 0,C 180,E1 -29171.915,E2 -29171.915} C_VEL
LIN {X 0,Y 143.447,Z 678.197,A -85,B 0,C 180,E1 -29172.37,E2 -29172.37} C_VEL
LIN {X 0,Y 138.845,Z 689.234,A -85,B 0,C 180,E1 -29173.001,E2 -29173.001} C_VEL
LIN {X 0,Y 133.852,Z 699.146,A -85,B 0,C 180,E1 -29173.752,E2 -29173.752} C_VEL
LIN {X 0,Y 128.07,Z 708.863,A -85,B 0,C 180,E1 -29174.722,E2 -29174.722} C_VEL
LIN {X 0,Y 121.506,Z 718.274,A -85,B 0,C 180,E1 -29175.934,E2 -29175.934} C_VEL
LIN {X 0,Y 114.251,Z 727.291,A -85,B 0,C 180,E1 -29177.553,E2 -29177.553} C_VEL
LIN {X 0,Y 108.219,Z 733.951,A -85,B 0,C 180,E1 -29179.109,E2 -29179.109} C_VEL
LIN {X 0,Y 100.075,Z 741.782,A -85,B 0,C 180,E1 -29181.489,E2 -29181.489} C_VEL
LIN {X 0,Y 92.394,Z 748.25,A -85,B 0,C 180,E1 -29184.11,E2 -29184.11} C_VEL
LIN {X 0,Y 83.546,Z 754.788,A -85,B 0,C 180,E1 -29187.963,E2 -29187.963} C_VEL
LIN {X 0,Y 75.182,Z 760.222,A -85,B 0,C 180,E1 -29192.722,E2 -29192.722} C_VEL
LIN {X 0,Y 67.448,Z 764.698,A -85,B 0,C 180,E1 -29198.7,E2 -29198.7} C_VEL
LIN {X 0,Y 60.68,Z 768.226,A -85,B 0,C 180,E1 -29205.98,E2 -29205.98} C_VEL
LIN {X 0,Y 56.761,Z 770.173,A -85,B 0,C 180,E1 -29211.752,E2 -29211.752} C_VEL
LIN {X 0,Y 50.937,Z 772.878,A -85,B 0,C 180,E1 -29225.549,E2 -29225.549} C_VEL
LIN {X 0,Y 48.396,Z 774.194,A -85,B 0,C 180,E1 -29241.65,E2 -29241.65} C_VEL
LIN {X 0,Y 48.368,Z 774.457,A -85,B 0,C 180,E1 -29250,E2 -29250} C_VEL
LIN {X 0,Y 49.248,Z 773.708,A -85,B 0,C 180,E1 -29266.583,E2 -29266.583} C_VEL
LIN {X 0,Y 50.937,Z 772.878,A -85,B 0,C 180,E1 -29274.451,E2 -29274.451} C_VEL
LIN {X 0,Y 56.758,Z 770.173,A -85,B 0,C 180,E1 -29288.251,E2 -29288.251} C_VEL
LIN {X 0,Y 62.846,Z 767.207,A -85,B 0,C 180,E1 -29296.625,E2 -29296.625} C_VEL
LIN {X 0,Y 69.959,Z 763.372,A -85,B 0,C 180,E1 -29303.481,E2 -29303.481} C_VEL
LIN {X 0,Y 77.909,Z 758.606,A -85,B 0,C 180,E1 -29308.976,E2 -29308.976} C_VEL
LIN {X 0,Y 87.902,Z 751.661,A -85,B 0,C 180,E1 -29314.086,E2 -29314.086} C_VEL
LIN {X 0,Y 96.987,Z 744.455,A -85,B 0,C 180,E1 -29317.502,E2 -29317.502} C_VEL
LIN {X 0,Y 104.774,Z 737.387,A -85,B 0,C 180,E1 -29319.895,E2 -29319.895} C_VEL
LIN {X 0,Y 112.679,Z 729.111,A -85,B 0,C 180,E1 -29322.017,E2 -29322.017} C_VEL
LIN {X 0,Y 119.906,Z 720.394,A -85,B 0,C 180,E1 -29323.691,E2 -29323.691} C_VEL
LIN {X 0,Y 126.445,Z 711.344,A -85,B 0,C 180,E1 -29324.952,E2 -29324.952} C_VEL
LIN {X 0,Y 132.196,Z 702.073,A -85,B 0,C 180,E1 -29325.98,E2 -29325.98} C_VEL
LIN {X 0,Y 137.167,Z 692.737,A -85,B 0,C 180,E1 -29326.774,E2 -29326.774} C_VEL
LIN {X 0,Y 141.768,Z 682.487,A -85,B 0,C 180,E1 -29327.412,E2 -29327.412} C_VEL
LIN {X 0,Y 145.443,Z 672.531,A -85,B 0,C 180,E1 -29327.891,E2 -29327.891} C_VEL
LIN {X 0,Y 148.82,Z 660.645,A -85,B 0,C 180,E1 -29328.339,E2 -29328.339} C_VEL
LIN {X 0,Y 151.176,Z 649.132,A -85,B 0,C 180,E1 -29328.626,E2 -29328.626} C_VEL
LIN {X 0,Y 152.451,Z 640.004,A -85,B 0,C 180,E1 -29328.89,E2 -29328.89} C_VEL
LIN {X 0,Y 151.343,Z 636.544,A -85,B 0,C 180,E1 -29332.326,E2 -29332.326} C_VEL
LIN {X 0,Y 150.792,Z 634.559,A -85,B 0,C 180,E1 -29334.952,E2 -29334.952} C_VEL
LIN {X 0,Y 150.467,Z 632.07,A -85,B 0,C 180,E1 -29339.999,E2 -29339.999} C_VEL
LIN {X 0,Y 151.065,Z 635.526,A -85,B 0,C 180,E1 -29346.867,E2 -29346.867} C_VEL
LIN {X 0,Y 152.017,Z 638.677,A -85,B 0,C 180,E1 -29350.308,E2 -29350.308} C_VEL
LIN {X 0,Y 153.25,Z 643.086,A -85,B 0,C 180,E1 -29353.706,E2 -29353.706} C_VEL
LIN {X 0,Y 154.663,Z 649.069,A -85,B 0,C 180,E1 -29357.033,E2 -29357.033} C_VEL
LIN {X 0,Y 155.553,Z 655.428,A -85,B 0,C 180,E1 -29359.697,E2 -29359.697} C_VEL
LIN {X 0,Y 156.199,Z 665.699,A -85,B 0,C 180,E1 -29363.183,E2 -29363.183} C_VEL
LIN {X 0,Y 157.03,Z 676.758,A -85,B 0,C 180,E1 -29367.305,E2 -29367.305} C_VEL
LIN {X 0,Y 158.241,Z 686.664,A -85,B 0,C 180,E1 -29371.455,E2 -29371.455} C_VEL
LIN {X 0,Y 160.137,Z 695.912,A -85,B 0,C 180,E1 -29375.808,E2 -29375.808} C_VEL
LIN {X 0,Y 161.43,Z 700.487,A -85,B 0,C 180,E1 -29378.112,E2 -29378.112} C_VEL
LIN {X 0,Y 162.075,Z 704.117,A -85,B 0,C 180,E1 -29379.751,E2 -29379.751} C_VEL
LIN {X 0,Y 161.824,Z 715.927,A -85,B 0,C 180,E1 -29384.477,E2 -29384.477} C_VEL
LIN {X 0,Y 162.736,Z 719.732,A -85,B 0,C 180,E1 -29386.465,E2 -29386.465} C_VEL
LIN {X 0,Y 162.998,Z 720.177,A -85,B 0,C 180,E1 -29386.757,E2 -29386.757} C_VEL
LIN {X 0,Y 170.604,Z 729.743,A -85,B 0,C 180,E1 -29393.444,E2 -29393.444} C_VEL
LIN {X 0,Y 179.838,Z 737.456,A -85,B 0,C 180,E1 -29399.286,E2 -29399.286} C_VEL
LIN {X 0,Y 190.789,Z 743.835,A -85,B 0,C 180,E1 -29404.485,E2 -29404.485} C_VEL
LIN {X 0,Y 205.431,Z 750.258,A -85,B 0,C 180,E1 -29409.995,E2 -29409.995} C_VEL
LIN {X 0,Y 213.897,Z 753.452,A -85,B 0,C 180,E1 -29412.8,E2 -29412.8} C_VEL
LIN {X 0,Y 224.363,Z 757.126,A -85,B 0,C 180,E1 -29416.176,E2 -29416.176} C_VEL
LIN {X 0,Y 229.884,Z 759.069,A -85,B 0,C 180,E1 -29418.037,E2 -29418.037} C_VEL
LIN {X 0,Y 235.455,Z 761.003,A -85,B 0,C 180,E1 -29420.059,E2 -29420.059} C_VEL
LIN {X 0,Y 239.071,Z 762.344,A -85,B 0,C 180,E1 -29421.548,E2 -29421.548} C_VEL
LIN {X 0,Y 242.71,Z 763.722,A -85,B 0,C 180,E1 -29423.349,E2 -29423.349} C_VEL
LIN {X 0,Y 246.656,Z 765.09,A -85,B 0,C 180,E1 -29425.745,E2 -29425.745} C_VEL
LIN {X 0,Y 247.932,Z 765.542,A -85,B 0,C 180,E1 -29426.75,E2 -29426.75} C_VEL
LIN {X 0,Y 249.533,Z 765.977,A -85,B 0,C 180,E1 -29428.386,E2 -29428.386} C_VEL
LIN {X 0,Y 250.486,Z 766.122,A -85,B 0,C 180,E1 -29430,E2 -29430} C_VEL
LIN {X 0,Y 249.539,Z 765.977,A -85,B 0,C 180,E1 -29431.614,E2 -29431.614} C_VEL
LIN {X 0,Y 247.959,Z 765.542,A -85,B 0,C 180,E1 -29433.25,E2 -29433.25} C_VEL
LIN {X 0,Y 245.571,Z 764.787,A -85,B 0,C 180,E1 -29434.925,E2 -29434.925} C_VEL
LIN {X 0,Y 242.738,Z 763.721,A -85,B 0,C 180,E1 -29436.65,E2 -29436.65} C_VEL
LIN {X 0,Y 239.066,Z 762.344,A -85,B 0,C 180,E1 -29438.452,E2 -29438.452} C_VEL
LIN {X 0,Y 234.359,Z 760.627,A -85,B 0,C 180,E1 -29440.365,E2 -29440.365} C_VEL
LIN {X 0,Y 228.505,Z 758.601,A -85,B 0,C 180,E1 -29442.433,E2 -29442.433} C_VEL
LIN {X 0,Y 221.709,Z 756.23,A -85,B 0,C 180,E1 -29444.69,E2 -29444.69} C_VEL
LIN {X 0,Y 213.514,Z 753.29,A -85,B 0,C 180,E1 -29447.342,E2 -29447.342} C_VEL
LIN {X 0,Y 200.506,Z 748.272,A -85,B 0,C 180,E1 -29451.745,E2 -29451.745} C_VEL
LIN {X 0,Y 186.53,Z 741.599,A -85,B 0,C 180,E1 -29457.402,E2 -29457.402} C_VEL
LIN {X 0,Y 175.963,Z 734.54,A -85,B 0,C 180,E1 -29462.995,E2 -29462.995} C_VEL
LIN {X 0,Y 167.522,Z 726.353,A -85,B 0,C 180,E1 -29468.997,E2 -29468.997} C_VEL
LIN {X 0,Y 161.625,Z 717.922,A -85,B 0,C 180,E1 -29474.715,E2 -29474.715} C_VEL
LIN {X 0,Y 157.556,Z 708.979,A -85,B 0,C 180,E1 -29480.264,E2 -29480.264} C_VEL
LIN {X 0,Y 155.023,Z 699.626,A -85,B 0,C 180,E1 -29485.48,E2 -29485.48} C_VEL
LIN {X 0,Y 153.614,Z 689.749,A -85,B 0,C 180,E1 -29490.372,E2 -29490.372} C_VEL
LIN {X 0,Y 153.02,Z 679.756,A -85,B 0,C 180,E1 -29494.733,E2 -29494.733} C_VEL
LIN {X 0,Y 152.903,Z 670.156,A -85,B 0,C 180,E1 -29498.427,E2 -29498.427} C_VEL
LIN {X 0,Y 152.793,Z 659.668,A -85,B 0,C 180,E1 -29502.186,E2 -29502.186} C_VEL
LIN {X 0,Y 152.245,Z 653.652,A -85,B 0,C 180,E1 -29504.867,E2 -29504.867} C_VEL
LIN {X 0,Y 151.392,Z 648.485,A -85,B 0,C 180,E1 -29507.983,E2 -29507.983} C_VEL
LIN {X 0,Y 150.543,Z 644.713,A -85,B 0,C 180,E1 -29511.105,E2 -29511.105} C_VEL
LIN {X 0,Y 149.868,Z 641.754,A -85,B 0,C 180,E1 -29514.62,E2 -29514.62} C_VEL
LIN {X 0,Y 149.585,Z 639.257,A -85,B 0,C 180,E1 -29520.001,E2 -29520.001} C_VEL
LIN {X 0,Y 150.023,Z 642.325,A -85,B 0,C 180,E1 -29525.841,E2 -29525.841} C_VEL
LIN {X 0,Y 150.597,Z 644.838,A -85,B 0,C 180,E1 -29528.602,E2 -29528.602} C_VEL
LIN {X 0,Y 148.243,Z 657.485,A -85,B 0,C 180,E1 -29528.889,E2 -29528.889} C_VEL
LIN {X 0,Y 145.727,Z 667.222,A -85,B 0,C 180,E1 -29529.184,E2 -29529.184} C_VEL
LIN {X 0,Y 141.669,Z 679.071,A -85,B 0,C 180,E1 -29529.617,E2 -29529.617} C_VEL
LIN {X 0,Y 137.423,Z 689.036,A -85,B 0,C 180,E1 -29530.118,E2 -29530.118} C_VEL
LIN {X 0,Y 132.344,Z 698.948,A -85,B 0,C 180,E1 -29530.765,E2 -29530.765} C_VEL
LIN {X 0,Y 126.453,Z 708.665,A -85,B 0,C 180,E1 -29531.61,E2 -29531.61} C_VEL
LIN {X 0,Y 119.752,Z 718.076,A -85,B 0,C 180,E1 -29532.667,E2 -29532.667} C_VEL
LIN {X 0,Y 112.303,Z 727.092,A -85,B 0,C 180,E1 -29534.076,E2 -29534.076} C_VEL
LIN {X 0,Y 105.429,Z 734.395,A -85,B 0,C 180,E1 -29535.627,E2 -29535.627} C_VEL
LIN {X 0,Y 97.682,Z 741.583,A -85,B 0,C 180,E1 -29537.583,E2 -29537.583} C_VEL
LIN {X 0,Y 88.142,Z 749.188,A -85,B 0,C 180,E1 -29540.47,E2 -29540.47} C_VEL
LIN {X 0,Y 80.443,Z 754.589,A -85,B 0,C 180,E1 -29543.462,E2 -29543.462} C_VEL
LIN {X 0,Y 71.566,Z 760.022,A -85,B 0,C 180,E1 -29547.895,E2 -29547.895} C_VEL
LIN {X 0,Y 65.957,Z 763.172,A -85,B 0,C 180,E1 -29551.525,E2 -29551.525} C_VEL
LIN {X 0,Y 55.765,Z 768.026,A -85,B 0,C 180,E1 -29560.873,E2 -29560.873} C_VEL
LIN {X 0,Y 51.343,Z 769.974,A -85,B 0,C 180,E1 -29566.811,E2 -29566.811} C_VEL
LIN {X 0,Y 44.528,Z 772.678,A -85,B 0,C 180,E1 -29581.739,E2 -29581.739} C_VEL
LIN {X 0,Y 41.376,Z 773.996,A -85,B 0,C 180,E1 -29600.221,E2 -29600.221} C_VEL
LIN {X 0,Y 41.279,Z 774.26,A -85,B 0,C 180,E1 -29610,E2 -29610} C_VEL
LIN {X 0,Y 42.473,Z 773.51,A -85,B 0,C 180,E1 -29629.325,E2 -29629.325} C_VEL
LIN {X 0,Y 44.527,Z 772.678,A -85,B 0,C 180,E1 -29638.262,E2 -29638.262} C_VEL
LIN {X 0,Y 51.339,Z 769.974,A -85,B 0,C 180,E1 -29653.192,E2 -29653.192} C_VEL
LIN {X 0,Y 58.153,Z 767.007,A -85,B 0,C 180,E1 -29661.77,E2 -29661.77} C_VEL
LIN {X 0,Y 65.957,Z 763.172,A -85,B 0,C 180,E1 -29668.475,E2 -29668.475} C_VEL
LIN {X 0,Y 74.477,Z 758.406,A -85,B 0,C 180,E1 -29673.694,E2 -29673.694} C_VEL
LIN {X 0,Y 85.029,Z 751.462,A -85,B 0,C 180,E1 -29678.41,E2 -29678.41} C_VEL
LIN {X 0,Y 92.891,Z 745.593,A -85,B 0,C 180,E1 -29681.033,E2 -29681.033} C_VEL
LIN {X 0,Y 100.916,Z 738.749,A -85,B 0,C 180,E1 -29683.246,E2 -29683.246} C_VEL
LIN {X 0,Y 109.049,Z 730.73,A -85,B 0,C 180,E1 -29685.172,E2 -29685.172} C_VEL
LIN {X 0,Y 117.272,Z 721.254,A -85,B 0,C 180,E1 -29686.861,E2 -29686.861} C_VEL
LIN {X 0,Y 123.949,Z 712.385,A -85,B 0,C 180,E1 -29687.977,E2 -29687.977} C_VEL
LIN {X 0,Y 129.811,Z 703.338,A -85,B 0,C 180,E1 -29688.893,E2 -29688.893} C_VEL
LIN {X 0,Y 135.717,Z 692.539,A -85,B 0,C 180,E1 -29689.697,E2 -29689.697} C_VEL
LIN {X 0,Y 140.391,Z 682.289,A -85,B 0,C 180,E1 -29690.244,E2 -29690.244} C_VEL
LIN {X 0,Y 144.525,Z 671.022,A -85,B 0,C 180,E1 -29690.712,E2 -29690.712} C_VEL
LIN {X 0,Y 147.56,Z 660.407,A -85,B 0,C 180,E1 -29691.038,E2 -29691.038} C_VEL
LIN {X 0,Y 149.94,Z 648.935,A -85,B 0,C 180,E1 -29691.28,E2 -29691.28} C_VEL
LIN {X 0,Y 150.566,Z 644.815,A -85,B 0,C 180,E1 -29691.396,E2 -29691.396} C_VEL
LIN {X 0,Y 149.86,Z 641.586,A -85,B 0,C 180,E1 -29695.223,E2 -29695.223} C_VEL
LIN {X 0,Y 149.587,Z 639.244,A -85,B 0,C 180,E1 -29699.999,E2 -29699.999} C_VEL
LIN {X 0,Y 149.981,Z 642.331,A -85,B 0,C 180,E1 -29706.22,E2 -29706.22} C_VEL
LIN {X 0,Y 150.76,Z 645.749,A -85,B 0,C 180,E1 -29709.929,E2 -29709.929} C_VEL
LIN {X 0,Y 151.809,Z 650.533,A -85,B 0,C 180,E1 -29713.383,E2 -29713.383} C_VEL
LIN {X 0,Y 152.516,Z 656.269,A -85,B 0,C 180,E1 -29716.398,E2 -29716.398} C_VEL
LIN {X 0,Y 152.94,Z 662.208,A -85,B 0,C 180,E1 -29718.762,E2 -29718.762} C_VEL
LIN {X 0,Y 152.965,Z 674.585,A -85,B 0,C 180,E1 -29723.237,E2 -29723.237} C_VEL
LIN {X 0,Y 153.277,Z 684.547,A -85,B 0,C 180,E1 -29727.29,E2 -29727.29} C_VEL
LIN {X 0,Y 154.309,Z 695.399,A -85,B 0,C 180,E1 -29732.353,E2 -29732.353} C_VEL
LIN {X 0,Y 156.275,Z 704.938,A -85,B 0,C 180,E1 -29737.402,E2 -29737.402} C_VEL
LIN {X 0,Y 159.723,Z 714.36,A -85,B 0,C 180,E1 -29743,E2 -29743} C_VEL
LIN {X 0,Y 162.998,Z 720.177,A -85,B 0,C 180,E1 -29746.757,E2 -29746.757} C_VEL
LIN {X 0,Y 164.194,Z 723.16,A -85,B 0,C 180,E1 -29748.505,E2 -29748.505} C_VEL
LIN {X 0,Y 165.609,Z 732.983,A -85,B 0,C 180,E1 -29753.668,E2 -29753.668} C_VEL
LIN {X 0,Y 167.028,Z 735.626,A -85,B 0,C 180,E1 -29755.409,E2 -29755.409} C_VEL
LIN {X 0,Y 167.763,Z 736.335,A -85,B 0,C 180,E1 -29755.979,E2 -29755.979} C_VEL
LIN {X 0,Y 177.077,Z 742.883,A -85,B 0,C 180,E1 -29761.559,E2 -29761.559} C_VEL
LIN {X 0,Y 190.24,Z 749.286,A -85,B 0,C 180,E1 -29767.45,E2 -29767.45} C_VEL
LIN {X 0,Y 202.174,Z 753.789,A -85,B 0,C 180,E1 -29771.769,E2 -29771.769} C_VEL
LIN {X 0,Y 211.244,Z 756.785,A -85,B 0,C 180,E1 -29774.752,E2 -29774.752} C_VEL
LIN {X 0,Y 218.079,Z 758.894,A -85,B 0,C 180,E1 -29776.963,E2 -29776.963} C_VEL
LIN {X 0,Y 224.621,Z 760.9,A -85,B 0,C 180,E1 -29779.18,E2 -29779.18} C_VEL
LIN {X 0,Y 230.147,Z 762.597,A -85,B 0,C 180,E1 -29781.218,E2 -29781.218} C_VEL
LIN {X 0,Y 234.53,Z 763.948,A -85,B 0,C 180,E1 -29783.116,E2 -29783.116} C_VEL
LIN {X 0,Y 239.524,Z 765.493,A -85,B 0,C 180,E1 -29786.025,E2 -29786.025} C_VEL
LIN {X 0,Y 240.399,Z 765.752,A -85,B 0,C 180,E1 -29786.648,E2 -29786.648} C_VEL
LIN {X 0,Y 242.189,Z 766.179,A -85,B 0,C 180,E1 -29788.337,E2 -29788.337} C_VEL
LIN {X 0,Y 243.314,Z 766.322,A -85,B 0,C 180,E1 -29790,E2 -29790} C_VEL
LIN {X 0,Y 242.2,Z 766.178,A -85,B 0,C 180,E1 -29791.663,E2 -29791.663} C_VEL
LIN {X 0,Y 240.412,Z 765.753,A -85,B 0,C 180,E1 -29793.352,E2 -29793.352} C_VEL
LIN {X 0,Y 237.701,Z 765.006,A -85,B 0,C 180,E1 -29795.089,E2 -29795.089} C_VEL
LIN {X 0,Y 233.782,Z 763.715,A -85,B 0,C 180,E1 -29797.236,E2 -29797.236} C_VEL
LIN {X 0,Y 228.079,Z 761.92,A -85,B 0,C 180,E1 -29799.59,E2 -29799.59} C_VEL
LIN {X 0,Y 222.403,Z 760.221,A -85,B 0,C 180,E1 -29801.596,E2 -29801.596} C_VEL
LIN {X 0,Y 216.794,Z 758.48,A -85,B 0,C 180,E1 -29803.464,E2 -29803.464} C_VEL
LIN {X 0,Y 205.801,Z 754.99,A -85,B 0,C 180,E1 -29807.027,E2 -29807.027} C_VEL
LIN {X 0,Y 193.552,Z 750.607,A -85,B 0,C 180,E1 -29811.291,E2 -29811.291} C_VEL
LIN {X 0,Y 180.794,Z 744.892,A -85,B 0,C 180,E1 -29816.613,E2 -29816.613} C_VEL
LIN {X 0,Y 172.337,Z 739.815,A -85,B 0,C 180,E1 -29821.089,E2 -29821.089} C_VEL
LIN {X 0,Y 163.869,Z 732.76,A -85,B 0,C 180,E1 -29826.9,E2 -29826.9} C_VEL
LIN {X 0,Y 158.221,Z 725.781,A -85,B 0,C 180,E1 -29832.218,E2 -29832.218} C_VEL
LIN {X 0,Y 154.052,Z 718.375,A -85,B 0,C 180,E1 -29837.503,E2 -29837.503} C_VEL
LIN {X 0,Y 151.075,Z 709.414,A -85,B 0,C 180,E1 -29843.25,E2 -29843.25} C_VEL
LIN {X 0,Y 149.659,Z 700.955,A -85,B 0,C 180,E1 -29848.111,E2 -29848.111} C_VEL
LIN {X 0,Y 149.143,Z 691.814,A -85,B 0,C 180,E1 -29852.756,E2 -29852.756} C_VEL
LIN {X 0,Y 149.246,Z 682.168,A -85,B 0,C 180,E1 -29857.091,E2 -29857.091} C_VEL
LIN {X 0,Y 149.784,Z 670.766,A -85,B 0,C 180,E1 -29861.537,E2 -29861.537} C_VEL
LIN {X 0,Y 150.103,Z 663.269,A -85,B 0,C 180,E1 -29864.383,E2 -29864.383} C_VEL
LIN {X 0,Y 149.82,Z 658.008,A -85,B 0,C 180,E1 -29866.957,E2 -29866.957} C_VEL
LIN {X 0,Y 149.348,Z 653.242,A -85,B 0,C 180,E1 -29870.181,E2 -29870.181} C_VEL
LIN {X 0,Y 148.894,Z 650.08,A -85,B 0,C 180,E1 -29873.267,E2 -29873.267} C_VEL
LIN {X 0,Y 148.617,Z 648.367,A -85,B 0,C 180,E1 -29875.637,E2 -29875.637} C_VEL
LIN {X 0,Y 148.572,Z 646.385,A -85,B 0,C 180,E1 -29880.001,E2 -29880.001} C_VEL
LIN {X 0,Y 148.775,Z 649.059,A -85,B 0,C 180,E1 -29885.117,E2 -29885.117} C_VEL
LIN {X 0,Y 148.878,Z 649.749,A -85,B 0,C 180,E1 -29885.953,E2 -29885.953} C_VEL
LIN {X 0,Y 145.683,Z 664.074,A -85,B 0,C 180,E1 -29886.313,E2 -29886.313} C_VEL
LIN {X 0,Y 141.089,Z 677.801,A -85,B 0,C 180,E1 -29886.728,E2 -29886.728} C_VEL
LIN {X 0,Y 136.356,Z 688.838,A -85,B 0,C 180,E1 -29887.182,E2 -29887.182} C_VEL
LIN {X 0,Y 131.204,Z 698.75,A -85,B 0,C 180,E1 -29887.721,E2 -29887.721} C_VEL
LIN {X 0,Y 125.217,Z 708.467,A -85,B 0,C 180,E1 -29888.425,E2 -29888.425} C_VEL
LIN {X 0,Y 118.397,Z 717.878,A -85,B 0,C 180,E1 -29889.309,E2 -29889.309} C_VEL
LIN {X 0,Y 110.782,Z 726.892,A -85,B 0,C 180,E1 -29890.487,E2 -29890.487} C_VEL
LIN {X 0,Y 103.021,Z 734.864,A -85,B 0,C 180,E1 -29891.973,E2 -29891.973} C_VEL
LIN {X 0,Y 94.112,Z 742.72,A -85,B 0,C 180,E1 -29893.886,E2 -29893.886} C_VEL
LIN {X 0,Y 85.911,Z 748.989,A -85,B 0,C 180,E1 -29896.014,E2 -29896.014} C_VEL
LIN {X 0,Y 77.867,Z 754.389,A -85,B 0,C 180,E1 -29898.618,E2 -29898.618} C_VEL
LIN {X 0,Y 68.517,Z 759.823,A -85,B 0,C 180,E1 -29902.611,E2 -29902.611} C_VEL
LIN {X 0,Y 59.604,Z 764.274,A -85,B 0,C 180,E1 -29907.84,E2 -29907.84} C_VEL
LIN {X 0,Y 51.377,Z 767.827,A -85,B 0,C 180,E1 -29914.841,E2 -29914.841} C_VEL
LIN {X 0,Y 46.397,Z 769.775,A -85,B 0,C 180,E1 -29920.768,E2 -29920.768} C_VEL
LIN {X 0,Y 38.387,Z 772.479,A -85,B 0,C 180,E1 -29936.686,E2 -29936.686} C_VEL
LIN {X 0,Y 34.378,Z 773.797,A -85,B 0,C 180,E1 -29958.204,E2 -29958.204} C_VEL
LIN {X 0,Y 34.164,Z 774.061,A -85,B 0,C 180,E1 -29970,E2 -29970} C_VEL
LIN {X 0,Y 35.81,Z 773.31,A -85,B 0,C 180,E1 -29993.111,E2 -29993.111} C_VEL
LIN {X 0,Y 38.387,Z 772.479,A -85,B 0,C 180,E1 -30003.315,E2 -30003.315} C_VEL
LIN {X 0,Y 46.393,Z 769.775,A -85,B 0,C 180,E1 -30019.238,E2 -30019.238} C_VEL
LIN {X 0,Y 54.01,Z 766.807,A -85,B 0,C 180,E1 -30027.756,E2 -30027.756} C_VEL
LIN {X 0,Y 62.519,Z 762.973,A -85,B 0,C 180,E1 -30034.064,E2 -30034.064} C_VEL
LIN {X 0,Y 71.591,Z 758.207,A -85,B 0,C 180,E1 -30038.84,E2 -30038.84} C_VEL
LIN {X 0,Y 82.67,Z 751.263,A -85,B 0,C 180,E1 -30043.014,E2 -30043.014} C_VEL
LIN {X 0,Y 90.827,Z 745.394,A -85,B 0,C 180,E1 -30045.284,E2 -30045.284} C_VEL
LIN {X 0,Y 99.102,Z 738.55,A -85,B 0,C 180,E1 -30047.183,E2 -30047.183} C_VEL
LIN {X 0,Y 107.442,Z 730.531,A -85,B 0,C 180,E1 -30048.86,E2 -30048.86} C_VEL
LIN {X 0,Y 115.865,Z 721.056,A -85,B 0,C 180,E1 -30050.283,E2 -30050.283} C_VEL
LIN {X 0,Y 122.664,Z 712.186,A -85,B 0,C 180,E1 -30051.232,E2 -30051.232} C_VEL
